// TwinCAT 3 PLC project PLC
// ProgramVersion: 3.1.4023.0
// libraries:
//   Tc2_Standard, * (Beckhoff Automation GmbH)
//   Tc2_System, * (Beckhoff Automation GmbH)
//   Tc3_Module, * (Beckhoff Automation GmbH)
// project tree:
//   / PlcTask.TcTTO
//   POUs/ MAIN.TcPOU
//   DUTs/IO/PdoEntries/ Status_3E6F3FF3.TcDUT, Control_6EF2C5D0.TcDUT, Status_237FCB0F.TcDUT, Setting_24C04940.TcDUT, Ctrl_56BB2DF2.TcDUT, Status_51F0A924.TcDUT, Settings_24C04940.TcDUT, Control_18D542D9.TcDUT, Status_396FCBA0.TcDUT, U1_STATUS_B0753356.TcDUT, U1_SAMPLES_2D13B74B.TcDUT, I1_STATUS_B0753356.TcDUT, I1_SAMPLES_2D13B74B.TcDUT, U2_STATUS_B0753356.TcDUT, U2_SAMPLES_2D13B74B.TcDUT, I2_STATUS_B0753356.TcDUT, I2_SAMPLES_2D13B74B.TcDUT, U3_STATUS_B0753356.TcDUT, U3_SAMPLES_2D13B74B.TcDUT, I3_STATUS_B0753356.TcDUT, I3_SAMPLES_2D13B74B.TcDUT, FSOE_31BB7F2A.TcDUT, FSOE_3C294B21.TcDUT, FSOE_13BCEA3F.TcDUT, FSOE_6A82EB93.TcDUT, FSOE_BB3344D6.TcDUT
//   DUTs/IO/PDOs/ InfoData_6F19DB2B.TcDUT, Channel_830843C1.TcDUT, Channel_42CA91F7.TcDUT, WcState_9091E0EB.TcDUT, DO_Diag_Inputs_CC455148.TcDUT, DO_Diag_Inputs_212B82C1.TcDUT, DO_Inputs_Device_AF161A9E.TcDUT, DO_Outputs_28AC1A9E.TcDUT, DO_Outputs_Device_36A5EF17.TcDUT, InfoData_32EB74EA.TcDUT, InfoData_0A66F009.TcDUT, ENC_Inputs_B3536485.TcDUT, ENC_Inputs_24B63C53.TcDUT, ENC_Outputs_21E2D14D.TcDUT, Ch1_CycleCount_9DBE2BC5.TcDUT, Ch1_Input_FFC4CE24.TcDUT, EMPTY_STRUCTURE.TcDUT, Ch2_CycleCount_976A51B5.TcDUT, Ch2_Input_78ADA90C.TcDUT, NextSync1Time_EE185E17.TcDUT, InfoData_A7436BC6.TcDUT, CycCount0_2C233804.TcDUT, Sample_0023574C.TcDUT, CycCount1_2C233804.TcDUT, Sample_07D5B44A.TcDUT, WcState_0B2B16F9.TcDUT, CycCount0_AF431CE0.TcDUT, CycCount1_A8B5FFE6.TcDUT, StartTimeNextOutput_228767F4.TcDUT, SAI_Inputs_3A838E11.TcDUT, SAI_Range_C3200E78.TcDUT, SAI_Range_3710D747.TcDUT, SAI_Inputs_84B29FE9.TcDUT, SAI_Range_BDBF6DA9.TcDUT, SAI_Range_2A187FC5.TcDUT, Channel_B90637B9.TcDUT, Channel_C6781B15.TcDUT, ENC_Inputs_3399C5AA.TcDUT, ENC_Outputs_2E45048F.TcDUT, ENC_Inputs_561E041F.TcDUT, ENC_Inputs_F139456B.TcDUT, ENC_Outputs_6FDDC669.TcDUT, L1_Voltage_Status_784F03AD.TcDUT, L1_Voltage_Samples_ED678DEE.TcDUT, L1_Current_Samples_89E07818.TcDUT, L1_Current_Samples_3209B12F.TcDUT, L2_Voltage_Status_0626A010.TcDUT, L2_Voltage_Samples_D91109BE.TcDUT, L2_Current_Status_F789DBA5.TcDUT, L2_Current_Samples_067F357F.TcDUT, L3_Voltage_Status_2C01C17B.TcDUT, L3_Voltage_Samples_CAC3758E.TcDUT, L3_Current_Status_DDAEBACE.TcDUT, L3_Current_Samples_15AD494F.TcDUT, AI_Timestamp_NextSync1Time_9AFDC275.TcDUT, AI_CycleCount_B1A935A2.TcDUT, InfoData_BEF6B88E.TcDUT, Digital_BD004D6F.TcDUT, Encoder_Channel_2E4EA213.TcDUT, Digital_A7E1DFAB.TcDUT, Analog_Channel_5F9B7EA6.TcDUT, Encoder_Channel_B7999E14.TcDUT, DeviceMain_Outputs_650F3486.TcDUT, FSoE_Slave_Connection_1_Slave_Message_330A35E4.TcDUT, Standard_Inputdata_FDD1436A.TcDUT, FSLOGIC_Inputs_CD3F9A93.TcDUT, FSoE_Slave_Connection_1_Master_Message_7109E4F0.TcDUT, Standard_Outputdata_59C030BE.TcDUT, Ch_A_AxisMain_Inputs_DC14661D.TcDUT, Ch_A_AxisMain_Outputs_A99AE12E.TcDUT, Ch_A_Interpolator_Outputs_462A5F1D.TcDUT, Ch_A_PositionControl_Inputs_8CB0F55A.TcDUT, WcState_B516A264.TcDUT, InfoData_358A59CF.TcDUT, Device_6E257577.TcDUT, Device_Safety_C21945A1.TcDUT, Ch_A_1FF86D85.TcDUT, Ch_A_AxisMain_Inputs_BA7CE8DB.TcDUT, Ch_A_D18C6F16.TcDUT, Ch_B_AxisMain_Inputs_A10B23CB.TcDUT, Ch_B_AxisMain_Outputs_526A47F8.TcDUT, Ch_B_Interpolator_Outputs_F819AE72.TcDUT, Ch_B_PositionControl_Inputs_C884000A.TcDUT, InfoData_386C00A5.TcDUT, Ch_B_5E084BAA.TcDUT, Ch_B_AxisMain_Inputs_3D4AF970.TcDUT, Ch_B_647F9A0C.TcDUT, InfoData_E68C61CD.TcDUT, InfoData_2A97D6CF.TcDUT, Inputs_25A0042B.TcDUT, Outputs_2397A10E.TcDUT
//   DUTs/IO/Boxes/ EK1100_1FC0878B.TcDUT, EK1122_1FC0878B.TcDUT, EPP2339_8DFD1558.TcDUT, EPP2349_8DFD1558.TcDUT, EP2316_3C060514.TcDUT, EP2338_39FFBC52.TcDUT, EP2339_C2A6198C.TcDUT, EP2339_56BCD6FB.TcDUT, EJ5151_905C5FD8.TcDUT, EL1262_0FA571DE.TcDUT, EL2262_79C970B1.TcDUT, EL2262_147DB6E1.TcDUT, EL2262_9619875D.TcDUT, EL3681_02A14E64.TcDUT, EL3681_0095B62C.TcDUT, EL5101_127DF9F1.TcDUT, EL5151_84FDBA5C.TcDUT, EL5151_93354628.TcDUT, EL5151_905C5FD8.TcDUT, EL5151_4D0E77FC.TcDUT, EL3773_D0D76902.TcDUT, EM7004_866015E1.TcDUT, AX8108_8297A621.TcDUT, AX8108_F7A82895.TcDUT, AX8118_8297A621.TcDUT, AX8118_F7A82895.TcDUT, AX8206_63F473B4.TcDUT, AX8206_FA9FF81E.TcDUT, AMP8000_F7A82895.TcDUT
//   DUTs/IO/Devices/ SyncUnitTask_2D604ED5.TcDUT, SyncUnitTasks_6FEB8257.TcDUT, SyncUnits_99E584AF.TcDUT
//   DUTs/IO/Topology/ boxesEK1122_B55A8AA2.TcDUT, boxes_17897972.TcDUT, EtherCAT_Master_Duplicates_CB89F35C.TcDUT
//   DUTs/IO/Base/ EtcSlaveBase_82538BE2.TcDUT, EtcSlaveBase_82538BE2.TcDUT, EtcSlaveBase_82538BE2.TcDUT, EtcSlaveTerminalBase_947E5A46.TcDUT, EtcSlaveBoxBase_77A0E4A7.TcDUT, EtcSlaveEndTerminalBase_866C7F0C.TcDUT, InputBase_8311D824.TcDUT, OutputBase_10CEE7DE.TcDUT, EtcMasterBase_62654B43.TcDUT
//   GVLs/ GVL_iXlinker.TcGVL

CONFIGURATION PLC
    RESOURCE PLC ON TwinCAT3
        TASK PlcTask(INTERVAL := T#10ms, PRIORITY := 20);
        PROGRAM MAIN WITH PlcTask : MAIN;
    END_RESOURCE
END_CONFIGURATION

// ---- DUTs/IO/PdoEntries/Status_3E6F3FF3.TcDUT
{attribute 'GeneratedUsingTerminal: EJ5151-0000-0016'}
{attribute addProperty BoxType "EJ5151-0000-0016"}
{attribute addProperty Id "Latch_C_validBOOL1Latch_extern_validBOOL1Set_counter_doneBOOL1Extrapolation_stallBOOL1Status_of_input_ABOOL1Status_of_input_BBOOL1Status_of_input_CBOOL1Status_of_extern_latchBOOL1Sync_errorBOOL1TxPDO_ToggleBOOL1"}
{attribute addProperty CRC "1047478259"}
{attribute addProperty Size "10"}
TYPE Status_3E6F3FF3 :
STRUCT
	{attribute addProperty Name "Latch_C_valid"}
	Latch_C_valid : BOOL;
	{attribute addProperty Name "Latch_extern_valid"}
	Latch_extern_valid : BOOL;
	{attribute addProperty Name "Set_counter_done"}
	Set_counter_done : BOOL;
	{attribute addProperty Name "Extrapolation_stall"}
	Extrapolation_stall : BOOL;
	{attribute addProperty Name "Status_of_input_A"}
	Status_of_input_A : BOOL;
	{attribute addProperty Name "Status_of_input_B"}
	Status_of_input_B : BOOL;
	{attribute addProperty Name "Status_of_input_C"}
	Status_of_input_C : BOOL;
	{attribute addProperty Name "Status_of_extern_latch"}
	Status_of_extern_latch : BOOL;
	{attribute addProperty Name "Sync_error"}
	Sync_error : BOOL;
	{attribute addProperty Name "TxPDO_Toggle"}
	TxPDO_Toggle : BOOL;
END_STRUCT
END_TYPE

// ---- DUTs/IO/PdoEntries/Control_6EF2C5D0.TcDUT
{attribute 'GeneratedUsingTerminal: EJ5151-0000-0016'}
{attribute addProperty BoxType "EJ5151-0000-0016"}
{attribute addProperty Id "Enable_latch_CBOOL1Enable_latch_extern_on_positive_edgeBOOL1Set_counterBOOL1Enable_latch_extern_on_negative_edgeBOOL1"}
{attribute addProperty CRC "1861404112"}
{attribute addProperty Size "4"}
TYPE Control_6EF2C5D0 :
STRUCT
	{attribute addProperty Name "Enable_latch_C"}
	Enable_latch_C : BOOL;
	{attribute addProperty Name "Enable_latch_extern_on_positive_edge"}
	Enable_latch_extern_on_positive_edge : BOOL;
	{attribute addProperty Name "Set_counter"}
	Set_counter : BOOL;
	{attribute addProperty Name "Enable_latch_extern_on_negative_edge"}
	Enable_latch_extern_on_negative_edge : BOOL;
END_STRUCT
END_TYPE

// ---- DUTs/IO/PdoEntries/Status_237FCB0F.TcDUT
{attribute 'GeneratedUsingTerminal: EL3681-0000-0017'}
{attribute addProperty BoxType "EL3681-0000-0017"}
{attribute addProperty Id "UnderrangeBOOL1OverrangeBOOL1Extended_rangeBOOL1Data_InvalidBOOL1Range_InvalidBOOL1Autorange_enabledBOOL1ErrorBOOL1Calibration_in_progressBOOL1TxPDO_StateBOOL1TxPDO_ToggleBOOL1"}
{attribute addProperty CRC "595577615"}
{attribute addProperty Size "10"}
TYPE Status_237FCB0F :
STRUCT
	{attribute addProperty Name "Underrange"}
	Underrange : BOOL;
	{attribute addProperty Name "Overrange"}
	Overrange : BOOL;
	{attribute addProperty Name "Extended_range"}
	Extended_range : BOOL;
	{attribute addProperty Name "Data_Invalid"}
	Data_Invalid : BOOL;
	{attribute addProperty Name "Range_Invalid"}
	Range_Invalid : BOOL;
	{attribute addProperty Name "Autorange_enabled"}
	Autorange_enabled : BOOL;
	{attribute addProperty Name "Error"}
	Error : BOOL;
	{attribute addProperty Name "Calibration_in_progress"}
	Calibration_in_progress : BOOL;
	{attribute addProperty Name "TxPDO_State"}
	TxPDO_State : BOOL;
	{attribute addProperty Name "TxPDO_Toggle"}
	TxPDO_Toggle : BOOL;
END_STRUCT
END_TYPE

// ---- DUTs/IO/PdoEntries/Setting_24C04940.TcDUT
{attribute 'GeneratedUsingTerminal: EL3681-0000-0017'}
{attribute addProperty BoxType "EL3681-0000-0017"}
{attribute addProperty Id "ModeBYTE1RangeSINT1"}
{attribute addProperty CRC "616581440"}
{attribute addProperty Size "2"}
TYPE Setting_24C04940 :
STRUCT
	{attribute addProperty Name "Mode"}
	Mode : BYTE;
	{attribute addProperty Name "Range"}
	Range : SINT;
END_STRUCT
END_TYPE

// ---- DUTs/IO/PdoEntries/Ctrl_56BB2DF2.TcDUT
{attribute 'GeneratedUsingTerminal: EL3681-0000-0017'}
{attribute addProperty BoxType "EL3681-0000-0017"}
{attribute addProperty Id "Enable_autorangeBOOL1ModeBYTE1RangeSINT1"}
{attribute addProperty CRC "1455107570"}
{attribute addProperty Size "3"}
TYPE Ctrl_56BB2DF2 :
STRUCT
	{attribute addProperty Name "Enable_autorange"}
	Enable_autorange : BOOL;
	{attribute addProperty Name "Mode"}
	Mode : BYTE;
	{attribute addProperty Name "Range"}
	Range : SINT;
END_STRUCT
END_TYPE

// ---- DUTs/IO/PdoEntries/Status_51F0A924.TcDUT
{attribute 'GeneratedUsingTerminal: EL3681-0000-0018'}
{attribute addProperty BoxType "EL3681-0000-0018"}
{attribute addProperty Id "UnderrangeBOOL1OverrangeBOOL1Extended_rangeBOOL1Data_invalidBOOL1Range_invalidBOOL1Autorange_disabledBOOL1ErrorBOOL1Calibration_in_progressBOOL1TxPDO_StateBOOL1TxPDO_ToggleBOOL1"}
{attribute addProperty CRC "1374726436"}
{attribute addProperty Size "10"}
TYPE Status_51F0A924 :
STRUCT
	{attribute addProperty Name "Underrange"}
	Underrange : BOOL;
	{attribute addProperty Name "Overrange"}
	Overrange : BOOL;
	{attribute addProperty Name "Extended_range"}
	Extended_range : BOOL;
	{attribute addProperty Name "Data_invalid"}
	Data_invalid : BOOL;
	{attribute addProperty Name "Range_invalid"}
	Range_invalid : BOOL;
	{attribute addProperty Name "Autorange_disabled"}
	Autorange_disabled : BOOL;
	{attribute addProperty Name "Error"}
	Error : BOOL;
	{attribute addProperty Name "Calibration_in_progress"}
	Calibration_in_progress : BOOL;
	{attribute addProperty Name "TxPDO_State"}
	TxPDO_State : BOOL;
	{attribute addProperty Name "TxPDO_Toggle"}
	TxPDO_Toggle : BOOL;
END_STRUCT
END_TYPE

// ---- DUTs/IO/PdoEntries/Settings_24C04940.TcDUT
{attribute 'GeneratedUsingTerminal: EL3681-0000-0018'}
{attribute addProperty BoxType "EL3681-0000-0018"}
{attribute addProperty Id "ModeBYTE1RangeSINT1"}
{attribute addProperty CRC "616581440"}
{attribute addProperty Size "2"}
TYPE Settings_24C04940 :
STRUCT
	{attribute addProperty Name "Mode"}
	Mode : BYTE;
	{attribute addProperty Name "Range"}
	Range : SINT;
END_STRUCT
END_TYPE

// ---- DUTs/IO/PdoEntries/Control_18D542D9.TcDUT
{attribute 'GeneratedUsingTerminal: EL3681-0000-0018'}
{attribute addProperty BoxType "EL3681-0000-0018"}
{attribute addProperty Id "Disable_autorangeBOOL1Start_calibrationBOOL1ModeBYTE1RangeSINT1"}
{attribute addProperty CRC "416629465"}
{attribute addProperty Size "4"}
TYPE Control_18D542D9 :
STRUCT
	{attribute addProperty Name "Disable_autorange"}
	Disable_autorange : BOOL;
	{attribute addProperty Name "Start_calibration"}
	Start_calibration : BOOL;
	{attribute addProperty Name "Mode"}
	Mode : BYTE;
	{attribute addProperty Name "Range"}
	Range : SINT;
END_STRUCT
END_TYPE

// ---- DUTs/IO/PdoEntries/Status_396FCBA0.TcDUT
{attribute 'GeneratedUsingTerminal: EL5151-0000-0016'}
{attribute addProperty BoxType "EL5151-0000-0016"}
{attribute addProperty Id "Latch_C_validBOOL1Latch_extern_validBOOL1Set_counter_doneBOOL1Status_of_input_ABOOL1Status_of_input_BBOOL1Status_of_input_CBOOL1Status_of_extern_latchBOOL1TxPDO_ToggleBOOL1"}
{attribute addProperty CRC "963627936"}
{attribute addProperty Size "8"}
TYPE Status_396FCBA0 :
STRUCT
	{attribute addProperty Name "Latch_C_valid"}
	Latch_C_valid : BOOL;
	{attribute addProperty Name "Latch_extern_valid"}
	Latch_extern_valid : BOOL;
	{attribute addProperty Name "Set_counter_done"}
	Set_counter_done : BOOL;
	{attribute addProperty Name "Status_of_input_A"}
	Status_of_input_A : BOOL;
	{attribute addProperty Name "Status_of_input_B"}
	Status_of_input_B : BOOL;
	{attribute addProperty Name "Status_of_input_C"}
	Status_of_input_C : BOOL;
	{attribute addProperty Name "Status_of_extern_latch"}
	Status_of_extern_latch : BOOL;
	{attribute addProperty Name "TxPDO_Toggle"}
	TxPDO_Toggle : BOOL;
END_STRUCT
END_TYPE

// ---- DUTs/IO/PdoEntries/U1_STATUS_B0753356.TcDUT
{attribute 'GeneratedUsingTerminal: EL3773-0000-0016'}
{attribute addProperty BoxType "EL3773-0000-0016"}
{attribute addProperty Id "UnderrangeBOOL1OverrangeBOOL1Limit_1BYTE1Limit_2BYTE1ErrorBOOL1Sync_errorBOOL1TxPDO_StateBOOL1TxPDO_ToggleBOOL1"}
{attribute addProperty CRC "2960470870"}
{attribute addProperty Size "8"}
TYPE U1_STATUS_B0753356 :
STRUCT
	{attribute addProperty Name "Underrange"}
	Underrange : BOOL;
	{attribute addProperty Name "Overrange"}
	Overrange : BOOL;
	{attribute addProperty Name "Limit_1"}
	Limit_1 : BYTE;
	{attribute addProperty Name "Limit_2"}
	Limit_2 : BYTE;
	{attribute addProperty Name "Error"}
	Error : BOOL;
	{attribute addProperty Name "Sync_error"}
	Sync_error : BOOL;
	{attribute addProperty Name "TxPDO_State"}
	TxPDO_State : BOOL;
	{attribute addProperty Name "TxPDO_Toggle"}
	TxPDO_Toggle : BOOL;
END_STRUCT
END_TYPE

// ---- DUTs/IO/PdoEntries/U1_SAMPLES_2D13B74B.TcDUT
{attribute 'GeneratedUsingTerminal: EL3773-0000-0016'}
{attribute addProperty BoxType "EL3773-0000-0016"}
{attribute addProperty Id "Sample_1INT2Sample_2INT2Sample_3INT2Sample_4INT2Sample_5INT2Sample_6INT2Sample_7INT2Sample_8INT2Sample_9INT2Sample_10INT2"}
{attribute addProperty CRC "756266827"}
{attribute addProperty Size "20"}
TYPE U1_SAMPLES_2D13B74B :
STRUCT
	{attribute addProperty Name "Sample_1"}
	Sample_1 : INT;
	{attribute addProperty Name "Sample_2"}
	Sample_2 : INT;
	{attribute addProperty Name "Sample_3"}
	Sample_3 : INT;
	{attribute addProperty Name "Sample_4"}
	Sample_4 : INT;
	{attribute addProperty Name "Sample_5"}
	Sample_5 : INT;
	{attribute addProperty Name "Sample_6"}
	Sample_6 : INT;
	{attribute addProperty Name "Sample_7"}
	Sample_7 : INT;
	{attribute addProperty Name "Sample_8"}
	Sample_8 : INT;
	{attribute addProperty Name "Sample_9"}
	Sample_9 : INT;
	{attribute addProperty Name "Sample_10"}
	Sample_10 : INT;
END_STRUCT
END_TYPE

// ---- DUTs/IO/PdoEntries/I1_STATUS_B0753356.TcDUT
{attribute 'GeneratedUsingTerminal: EL3773-0000-0016'}
{attribute addProperty BoxType "EL3773-0000-0016"}
{attribute addProperty Id "UnderrangeBOOL1OverrangeBOOL1Limit_1BYTE1Limit_2BYTE1ErrorBOOL1Sync_errorBOOL1TxPDO_StateBOOL1TxPDO_ToggleBOOL1"}
{attribute addProperty CRC "2960470870"}
{attribute addProperty Size "8"}
TYPE I1_STATUS_B0753356 :
STRUCT
	{attribute addProperty Name "Underrange"}
	Underrange : BOOL;
	{attribute addProperty Name "Overrange"}
	Overrange : BOOL;
	{attribute addProperty Name "Limit_1"}
	Limit_1 : BYTE;
	{attribute addProperty Name "Limit_2"}
	Limit_2 : BYTE;
	{attribute addProperty Name "Error"}
	Error : BOOL;
	{attribute addProperty Name "Sync_error"}
	Sync_error : BOOL;
	{attribute addProperty Name "TxPDO_State"}
	TxPDO_State : BOOL;
	{attribute addProperty Name "TxPDO_Toggle"}
	TxPDO_Toggle : BOOL;
END_STRUCT
END_TYPE

// ---- DUTs/IO/PdoEntries/I1_SAMPLES_2D13B74B.TcDUT
{attribute 'GeneratedUsingTerminal: EL3773-0000-0016'}
{attribute addProperty BoxType "EL3773-0000-0016"}
{attribute addProperty Id "Sample_1INT2Sample_2INT2Sample_3INT2Sample_4INT2Sample_5INT2Sample_6INT2Sample_7INT2Sample_8INT2Sample_9INT2Sample_10INT2"}
{attribute addProperty CRC "756266827"}
{attribute addProperty Size "20"}
TYPE I1_SAMPLES_2D13B74B :
STRUCT
	{attribute addProperty Name "Sample_1"}
	Sample_1 : INT;
	{attribute addProperty Name "Sample_2"}
	Sample_2 : INT;
	{attribute addProperty Name "Sample_3"}
	Sample_3 : INT;
	{attribute addProperty Name "Sample_4"}
	Sample_4 : INT;
	{attribute addProperty Name "Sample_5"}
	Sample_5 : INT;
	{attribute addProperty Name "Sample_6"}
	Sample_6 : INT;
	{attribute addProperty Name "Sample_7"}
	Sample_7 : INT;
	{attribute addProperty Name "Sample_8"}
	Sample_8 : INT;
	{attribute addProperty Name "Sample_9"}
	Sample_9 : INT;
	{attribute addProperty Name "Sample_10"}
	Sample_10 : INT;
END_STRUCT
END_TYPE

// ---- DUTs/IO/PdoEntries/U2_STATUS_B0753356.TcDUT
{attribute 'GeneratedUsingTerminal: EL3773-0000-0016'}
{attribute addProperty BoxType "EL3773-0000-0016"}
{attribute addProperty Id "UnderrangeBOOL1OverrangeBOOL1Limit_1BYTE1Limit_2BYTE1ErrorBOOL1Sync_errorBOOL1TxPDO_StateBOOL1TxPDO_ToggleBOOL1"}
{attribute addProperty CRC "2960470870"}
{attribute addProperty Size "8"}
TYPE U2_STATUS_B0753356 :
STRUCT
	{attribute addProperty Name "Underrange"}
	Underrange : BOOL;
	{attribute addProperty Name "Overrange"}
	Overrange : BOOL;
	{attribute addProperty Name "Limit_1"}
	Limit_1 : BYTE;
	{attribute addProperty Name "Limit_2"}
	Limit_2 : BYTE;
	{attribute addProperty Name "Error"}
	Error : BOOL;
	{attribute addProperty Name "Sync_error"}
	Sync_error : BOOL;
	{attribute addProperty Name "TxPDO_State"}
	TxPDO_State : BOOL;
	{attribute addProperty Name "TxPDO_Toggle"}
	TxPDO_Toggle : BOOL;
END_STRUCT
END_TYPE

// ---- DUTs/IO/PdoEntries/U2_SAMPLES_2D13B74B.TcDUT
{attribute 'GeneratedUsingTerminal: EL3773-0000-0016'}
{attribute addProperty BoxType "EL3773-0000-0016"}
{attribute addProperty Id "Sample_1INT2Sample_2INT2Sample_3INT2Sample_4INT2Sample_5INT2Sample_6INT2Sample_7INT2Sample_8INT2Sample_9INT2Sample_10INT2"}
{attribute addProperty CRC "756266827"}
{attribute addProperty Size "20"}
TYPE U2_SAMPLES_2D13B74B :
STRUCT
	{attribute addProperty Name "Sample_1"}
	Sample_1 : INT;
	{attribute addProperty Name "Sample_2"}
	Sample_2 : INT;
	{attribute addProperty Name "Sample_3"}
	Sample_3 : INT;
	{attribute addProperty Name "Sample_4"}
	Sample_4 : INT;
	{attribute addProperty Name "Sample_5"}
	Sample_5 : INT;
	{attribute addProperty Name "Sample_6"}
	Sample_6 : INT;
	{attribute addProperty Name "Sample_7"}
	Sample_7 : INT;
	{attribute addProperty Name "Sample_8"}
	Sample_8 : INT;
	{attribute addProperty Name "Sample_9"}
	Sample_9 : INT;
	{attribute addProperty Name "Sample_10"}
	Sample_10 : INT;
END_STRUCT
END_TYPE

// ---- DUTs/IO/PdoEntries/I2_STATUS_B0753356.TcDUT
{attribute 'GeneratedUsingTerminal: EL3773-0000-0016'}
{attribute addProperty BoxType "EL3773-0000-0016"}
{attribute addProperty Id "UnderrangeBOOL1OverrangeBOOL1Limit_1BYTE1Limit_2BYTE1ErrorBOOL1Sync_errorBOOL1TxPDO_StateBOOL1TxPDO_ToggleBOOL1"}
{attribute addProperty CRC "2960470870"}
{attribute addProperty Size "8"}
TYPE I2_STATUS_B0753356 :
STRUCT
	{attribute addProperty Name "Underrange"}
	Underrange : BOOL;
	{attribute addProperty Name "Overrange"}
	Overrange : BOOL;
	{attribute addProperty Name "Limit_1"}
	Limit_1 : BYTE;
	{attribute addProperty Name "Limit_2"}
	Limit_2 : BYTE;
	{attribute addProperty Name "Error"}
	Error : BOOL;
	{attribute addProperty Name "Sync_error"}
	Sync_error : BOOL;
	{attribute addProperty Name "TxPDO_State"}
	TxPDO_State : BOOL;
	{attribute addProperty Name "TxPDO_Toggle"}
	TxPDO_Toggle : BOOL;
END_STRUCT
END_TYPE

// ---- DUTs/IO/PdoEntries/I2_SAMPLES_2D13B74B.TcDUT
{attribute 'GeneratedUsingTerminal: EL3773-0000-0016'}
{attribute addProperty BoxType "EL3773-0000-0016"}
{attribute addProperty Id "Sample_1INT2Sample_2INT2Sample_3INT2Sample_4INT2Sample_5INT2Sample_6INT2Sample_7INT2Sample_8INT2Sample_9INT2Sample_10INT2"}
{attribute addProperty CRC "756266827"}
{attribute addProperty Size "20"}
TYPE I2_SAMPLES_2D13B74B :
STRUCT
	{attribute addProperty Name "Sample_1"}
	Sample_1 : INT;
	{attribute addProperty Name "Sample_2"}
	Sample_2 : INT;
	{attribute addProperty Name "Sample_3"}
	Sample_3 : INT;
	{attribute addProperty Name "Sample_4"}
	Sample_4 : INT;
	{attribute addProperty Name "Sample_5"}
	Sample_5 : INT;
	{attribute addProperty Name "Sample_6"}
	Sample_6 : INT;
	{attribute addProperty Name "Sample_7"}
	Sample_7 : INT;
	{attribute addProperty Name "Sample_8"}
	Sample_8 : INT;
	{attribute addProperty Name "Sample_9"}
	Sample_9 : INT;
	{attribute addProperty Name "Sample_10"}
	Sample_10 : INT;
END_STRUCT
END_TYPE

// ---- DUTs/IO/PdoEntries/U3_STATUS_B0753356.TcDUT
{attribute 'GeneratedUsingTerminal: EL3773-0000-0016'}
{attribute addProperty BoxType "EL3773-0000-0016"}
{attribute addProperty Id "UnderrangeBOOL1OverrangeBOOL1Limit_1BYTE1Limit_2BYTE1ErrorBOOL1Sync_errorBOOL1TxPDO_StateBOOL1TxPDO_ToggleBOOL1"}
{attribute addProperty CRC "2960470870"}
{attribute addProperty Size "8"}
TYPE U3_STATUS_B0753356 :
STRUCT
	{attribute addProperty Name "Underrange"}
	Underrange : BOOL;
	{attribute addProperty Name "Overrange"}
	Overrange : BOOL;
	{attribute addProperty Name "Limit_1"}
	Limit_1 : BYTE;
	{attribute addProperty Name "Limit_2"}
	Limit_2 : BYTE;
	{attribute addProperty Name "Error"}
	Error : BOOL;
	{attribute addProperty Name "Sync_error"}
	Sync_error : BOOL;
	{attribute addProperty Name "TxPDO_State"}
	TxPDO_State : BOOL;
	{attribute addProperty Name "TxPDO_Toggle"}
	TxPDO_Toggle : BOOL;
END_STRUCT
END_TYPE

// ---- DUTs/IO/PdoEntries/U3_SAMPLES_2D13B74B.TcDUT
{attribute 'GeneratedUsingTerminal: EL3773-0000-0016'}
{attribute addProperty BoxType "EL3773-0000-0016"}
{attribute addProperty Id "Sample_1INT2Sample_2INT2Sample_3INT2Sample_4INT2Sample_5INT2Sample_6INT2Sample_7INT2Sample_8INT2Sample_9INT2Sample_10INT2"}
{attribute addProperty CRC "756266827"}
{attribute addProperty Size "20"}
TYPE U3_SAMPLES_2D13B74B :
STRUCT
	{attribute addProperty Name "Sample_1"}
	Sample_1 : INT;
	{attribute addProperty Name "Sample_2"}
	Sample_2 : INT;
	{attribute addProperty Name "Sample_3"}
	Sample_3 : INT;
	{attribute addProperty Name "Sample_4"}
	Sample_4 : INT;
	{attribute addProperty Name "Sample_5"}
	Sample_5 : INT;
	{attribute addProperty Name "Sample_6"}
	Sample_6 : INT;
	{attribute addProperty Name "Sample_7"}
	Sample_7 : INT;
	{attribute addProperty Name "Sample_8"}
	Sample_8 : INT;
	{attribute addProperty Name "Sample_9"}
	Sample_9 : INT;
	{attribute addProperty Name "Sample_10"}
	Sample_10 : INT;
END_STRUCT
END_TYPE

// ---- DUTs/IO/PdoEntries/I3_STATUS_B0753356.TcDUT
{attribute 'GeneratedUsingTerminal: EL3773-0000-0016'}
{attribute addProperty BoxType "EL3773-0000-0016"}
{attribute addProperty Id "UnderrangeBOOL1OverrangeBOOL1Limit_1BYTE1Limit_2BYTE1ErrorBOOL1Sync_errorBOOL1TxPDO_StateBOOL1TxPDO_ToggleBOOL1"}
{attribute addProperty CRC "2960470870"}
{attribute addProperty Size "8"}
TYPE I3_STATUS_B0753356 :
STRUCT
	{attribute addProperty Name "Underrange"}
	Underrange : BOOL;
	{attribute addProperty Name "Overrange"}
	Overrange : BOOL;
	{attribute addProperty Name "Limit_1"}
	Limit_1 : BYTE;
	{attribute addProperty Name "Limit_2"}
	Limit_2 : BYTE;
	{attribute addProperty Name "Error"}
	Error : BOOL;
	{attribute addProperty Name "Sync_error"}
	Sync_error : BOOL;
	{attribute addProperty Name "TxPDO_State"}
	TxPDO_State : BOOL;
	{attribute addProperty Name "TxPDO_Toggle"}
	TxPDO_Toggle : BOOL;
END_STRUCT
END_TYPE

// ---- DUTs/IO/PdoEntries/I3_SAMPLES_2D13B74B.TcDUT
{attribute 'GeneratedUsingTerminal: EL3773-0000-0016'}
{attribute addProperty BoxType "EL3773-0000-0016"}
{attribute addProperty Id "Sample_1INT2Sample_2INT2Sample_3INT2Sample_4INT2Sample_5INT2Sample_6INT2Sample_7INT2Sample_8INT2Sample_9INT2Sample_10INT2"}
{attribute addProperty CRC "756266827"}
{attribute addProperty Size "20"}
TYPE I3_SAMPLES_2D13B74B :
STRUCT
	{attribute addProperty Name "Sample_1"}
	Sample_1 : INT;
	{attribute addProperty Name "Sample_2"}
	Sample_2 : INT;
	{attribute addProperty Name "Sample_3"}
	Sample_3 : INT;
	{attribute addProperty Name "Sample_4"}
	Sample_4 : INT;
	{attribute addProperty Name "Sample_5"}
	Sample_5 : INT;
	{attribute addProperty Name "Sample_6"}
	Sample_6 : INT;
	{attribute addProperty Name "Sample_7"}
	Sample_7 : INT;
	{attribute addProperty Name "Sample_8"}
	Sample_8 : INT;
	{attribute addProperty Name "Sample_9"}
	Sample_9 : INT;
	{attribute addProperty Name "Sample_10"}
	Sample_10 : INT;
END_STRUCT
END_TYPE

// ---- DUTs/IO/PdoEntries/FSOE_31BB7F2A.TcDUT
{attribute 'GeneratedUsingTerminal: AX8108-0100-0101-0101'}
{attribute addProperty BoxType "AX8108-0100-0101-0101"}
{attribute addProperty Id "FSoE_Slave_CmdUSINT1Axis_A_STOBOOL1Safe_Input_1BOOL1Safe_Input_2BOOL1Safe_Input_3BOOL1Safe_Input_4BOOL1Safe_Input_5BOOL1Safe_Input_6BOOL1Safe_Input_7BOOL1Axis_B_STOBOOL1Safe_Input_9BOOL1Safe_Input_10BOOL1Safe_Input_11BOOL1Safe_Input_12BOOL1Safe_Input_13BOOL1Safe_Input_14BOOL1Safe_Input_15BOOL1FSoE_Slave_CRC_0UINT2FSoE_Slave_ConnIDUINT2"}
{attribute addProperty CRC "834371370"}
{attribute addProperty Size "21"}
TYPE FSOE_31BB7F2A :
STRUCT
	{attribute addProperty Name "FSoE_Slave_Cmd"}
	FSoE_Slave_Cmd : USINT;
	{attribute addProperty Name "Axis_A_STO"}
	Axis_A_STO : BOOL;
	{attribute addProperty Name "Safe_Input_1"}
	Safe_Input_1 : BOOL;
	{attribute addProperty Name "Safe_Input_2"}
	Safe_Input_2 : BOOL;
	{attribute addProperty Name "Safe_Input_3"}
	Safe_Input_3 : BOOL;
	{attribute addProperty Name "Safe_Input_4"}
	Safe_Input_4 : BOOL;
	{attribute addProperty Name "Safe_Input_5"}
	Safe_Input_5 : BOOL;
	{attribute addProperty Name "Safe_Input_6"}
	Safe_Input_6 : BOOL;
	{attribute addProperty Name "Safe_Input_7"}
	Safe_Input_7 : BOOL;
	{attribute addProperty Name "Axis_B_STO"}
	Axis_B_STO : BOOL;
	{attribute addProperty Name "Safe_Input_9"}
	Safe_Input_9 : BOOL;
	{attribute addProperty Name "Safe_Input_10"}
	Safe_Input_10 : BOOL;
	{attribute addProperty Name "Safe_Input_11"}
	Safe_Input_11 : BOOL;
	{attribute addProperty Name "Safe_Input_12"}
	Safe_Input_12 : BOOL;
	{attribute addProperty Name "Safe_Input_13"}
	Safe_Input_13 : BOOL;
	{attribute addProperty Name "Safe_Input_14"}
	Safe_Input_14 : BOOL;
	{attribute addProperty Name "Safe_Input_15"}
	Safe_Input_15 : BOOL;
	{attribute addProperty Name "FSoE_Slave_CRC_0"}
	FSoE_Slave_CRC_0 : UINT;
	{attribute addProperty Name "FSoE_Slave_ConnID"}
	FSoE_Slave_ConnID : UINT;
END_STRUCT
END_TYPE

// ---- DUTs/IO/PdoEntries/FSOE_3C294B21.TcDUT
{attribute 'GeneratedUsingTerminal: AX8108-0100-0101-0101'}
{attribute addProperty BoxType "AX8108-0100-0101-0101"}
{attribute addProperty Id "Std_InputBOOL1Std_Input_1BOOL1Std_Input_2BOOL1Std_Input_3BOOL1Std_Input_4BOOL1Std_Input_5BOOL1Std_Input_6BOOL1Std_Input_7BOOL1"}
{attribute addProperty CRC "1009339169"}
{attribute addProperty Size "8"}
TYPE FSOE_3C294B21 :
STRUCT
	{attribute addProperty Name "Std_Input"}
	Std_Input : BOOL;
	{attribute addProperty Name "Std_Input_1"}
	Std_Input_1 : BOOL;
	{attribute addProperty Name "Std_Input_2"}
	Std_Input_2 : BOOL;
	{attribute addProperty Name "Std_Input_3"}
	Std_Input_3 : BOOL;
	{attribute addProperty Name "Std_Input_4"}
	Std_Input_4 : BOOL;
	{attribute addProperty Name "Std_Input_5"}
	Std_Input_5 : BOOL;
	{attribute addProperty Name "Std_Input_6"}
	Std_Input_6 : BOOL;
	{attribute addProperty Name "Std_Input_7"}
	Std_Input_7 : BOOL;
END_STRUCT
END_TYPE

// ---- DUTs/IO/PdoEntries/FSOE_13BCEA3F.TcDUT
{attribute 'GeneratedUsingTerminal: AX8108-0100-0101-0101'}
{attribute addProperty BoxType "AX8108-0100-0101-0101"}
{attribute addProperty Id "Safe_Logic_StateUSINT1Cycle_CounterUSINT1"}
{attribute addProperty CRC "331147839"}
{attribute addProperty Size "2"}
TYPE FSOE_13BCEA3F :
STRUCT
	{attribute addProperty Name "Safe_Logic_State"}
	Safe_Logic_State : USINT;
	{attribute addProperty Name "Cycle_Counter"}
	Cycle_Counter : USINT;
END_STRUCT
END_TYPE

// ---- DUTs/IO/PdoEntries/FSOE_6A82EB93.TcDUT
{attribute 'GeneratedUsingTerminal: AX8108-0100-0101-0101'}
{attribute addProperty BoxType "AX8108-0100-0101-0101"}
{attribute addProperty Id "FSoE_Master_CmdUSINT1Axis_A_STOBOOL1Safe_Output_1BOOL1Safe_Output_2BOOL1Safe_Output_3BOOL1Safe_Output_4BOOL1Safe_Output_5BOOL1Safe_Output_6BOOL1Safe_Output_7BOOL1Axis_B_STOBOOL1Safe_Output_9BOOL1Safe_Output_10BOOL1Safe_Output_11BOOL1Safe_Output_12BOOL1Safe_Output_13BOOL1Safe_Output_14BOOL1Safe_Output_15BOOL1FSoE_Master_CRC_0UINT2FSoE_Master_ConnIDUINT2"}
{attribute addProperty CRC "1786964883"}
{attribute addProperty Size "21"}
TYPE FSOE_6A82EB93 :
STRUCT
	{attribute addProperty Name "FSoE_Master_Cmd"}
	FSoE_Master_Cmd : USINT;
	{attribute addProperty Name "Axis_A_STO"}
	Axis_A_STO : BOOL;
	{attribute addProperty Name "Safe_Output_1"}
	Safe_Output_1 : BOOL;
	{attribute addProperty Name "Safe_Output_2"}
	Safe_Output_2 : BOOL;
	{attribute addProperty Name "Safe_Output_3"}
	Safe_Output_3 : BOOL;
	{attribute addProperty Name "Safe_Output_4"}
	Safe_Output_4 : BOOL;
	{attribute addProperty Name "Safe_Output_5"}
	Safe_Output_5 : BOOL;
	{attribute addProperty Name "Safe_Output_6"}
	Safe_Output_6 : BOOL;
	{attribute addProperty Name "Safe_Output_7"}
	Safe_Output_7 : BOOL;
	{attribute addProperty Name "Axis_B_STO"}
	Axis_B_STO : BOOL;
	{attribute addProperty Name "Safe_Output_9"}
	Safe_Output_9 : BOOL;
	{attribute addProperty Name "Safe_Output_10"}
	Safe_Output_10 : BOOL;
	{attribute addProperty Name "Safe_Output_11"}
	Safe_Output_11 : BOOL;
	{attribute addProperty Name "Safe_Output_12"}
	Safe_Output_12 : BOOL;
	{attribute addProperty Name "Safe_Output_13"}
	Safe_Output_13 : BOOL;
	{attribute addProperty Name "Safe_Output_14"}
	Safe_Output_14 : BOOL;
	{attribute addProperty Name "Safe_Output_15"}
	Safe_Output_15 : BOOL;
	{attribute addProperty Name "FSoE_Master_CRC_0"}
	FSoE_Master_CRC_0 : UINT;
	{attribute addProperty Name "FSoE_Master_ConnID"}
	FSoE_Master_ConnID : UINT;
END_STRUCT
END_TYPE

// ---- DUTs/IO/PdoEntries/FSOE_BB3344D6.TcDUT
{attribute 'GeneratedUsingTerminal: AX8108-0100-0101-0101'}
{attribute addProperty BoxType "AX8108-0100-0101-0101"}
{attribute addProperty Id "Std_OutputBOOL1Std_Output_1BOOL1Std_Output_2BOOL1Std_Output_3BOOL1Std_Output_4BOOL1Std_Output_5BOOL1Std_Output_6BOOL1Std_Output_7BOOL1"}
{attribute addProperty CRC "3140699350"}
{attribute addProperty Size "8"}
TYPE FSOE_BB3344D6 :
STRUCT
	{attribute addProperty Name "Std_Output"}
	Std_Output : BOOL;
	{attribute addProperty Name "Std_Output_1"}
	Std_Output_1 : BOOL;
	{attribute addProperty Name "Std_Output_2"}
	Std_Output_2 : BOOL;
	{attribute addProperty Name "Std_Output_3"}
	Std_Output_3 : BOOL;
	{attribute addProperty Name "Std_Output_4"}
	Std_Output_4 : BOOL;
	{attribute addProperty Name "Std_Output_5"}
	Std_Output_5 : BOOL;
	{attribute addProperty Name "Std_Output_6"}
	Std_Output_6 : BOOL;
	{attribute addProperty Name "Std_Output_7"}
	Std_Output_7 : BOOL;
END_STRUCT
END_TYPE

// ---- DUTs/IO/PDOs/InfoData_6F19DB2B.TcDUT
{attribute 'GeneratedUsingTerminal: EK1100-0000-0018'}
{attribute addProperty BoxType "EK1100-0000-0018"}
{attribute addProperty Id "StateAT %I*UINT2"}
{attribute addProperty CRC "1863965483"}
{attribute addProperty Size "2"}
TYPE InfoData_6F19DB2B :
STRUCT
	{attribute addProperty Name "State"}
	State AT %I* : UINT;
END_STRUCT
END_TYPE

// ---- DUTs/IO/PDOs/Channel_830843C1.TcDUT
{attribute 'GeneratedUsingTerminal: EPP2339-0021-0016'}
{attribute addProperty BoxType "EPP2339-0021-0016"}
{attribute addProperty Id "InputAT %I*BOOL1"}
{attribute addProperty CRC "2198356929"}
{attribute addProperty Size "1"}
TYPE Channel_830843C1 EXTENDS InputBase_8311D824 :
STRUCT
	{attribute addProperty Name "Input"}
	Input AT %I* : BOOL;
END_STRUCT
END_TYPE

// ---- DUTs/IO/PDOs/Channel_42CA91F7.TcDUT
{attribute 'GeneratedUsingTerminal: EPP2339-0021-0016'}
{attribute addProperty BoxType "EPP2339-0021-0016"}
{attribute addProperty Id "OutputAT %Q*BOOL1"}
{attribute addProperty CRC "1120571895"}
{attribute addProperty Size "1"}
TYPE Channel_42CA91F7 EXTENDS OutputBase_10CEE7DE :
STRUCT
	{attribute addProperty Name "Output"}
	Output AT %Q* : BOOL;
END_STRUCT
END_TYPE

// ---- DUTs/IO/PDOs/WcState_9091E0EB.TcDUT
{attribute 'GeneratedUsingTerminal: EPP2339-0021-0016'}
{attribute addProperty BoxType "EPP2339-0021-0016"}
{attribute addProperty Id "WcStateAT %I*BOOL1InputToggleAT %I*BOOL1"}
{attribute addProperty CRC "2425479403"}
{attribute addProperty Size "2"}
TYPE WcState_9091E0EB :
STRUCT
	{attribute addProperty Name "WcState"}
	WcState AT %I* : BOOL;
	{attribute addProperty Name "InputToggle"}
	InputToggle AT %I* : BOOL;
END_STRUCT
END_TYPE

// ---- DUTs/IO/PDOs/DO_Diag_Inputs_CC455148.TcDUT
{attribute 'GeneratedUsingTerminal: EP2316-0008-0017'}
{attribute addProperty BoxType "EP2316-0008-0017"}
{attribute addProperty Id "InputAT %I*ARRAY[0..7] OF BOOL8Sync_ErrorAT %I*BOOL1"}
{attribute addProperty CRC "2788215981"}
{attribute addProperty Size "9"}
TYPE DO_Diag_Inputs_CC455148 EXTENDS InputBase_8311D824 :
STRUCT
	{attribute addProperty Name "Input"}
	Input AT %I* : ARRAY[0..7] OF BOOL;
	{attribute addProperty Name "Sync_Error"}
	Sync_Error AT %I* : BOOL;
END_STRUCT
END_TYPE

// ---- DUTs/IO/PDOs/DO_Diag_Inputs_212B82C1.TcDUT
{attribute 'GeneratedUsingTerminal: EP2316-0008-0017'}
{attribute addProperty BoxType "EP2316-0008-0017"}
{attribute addProperty Id "Diag_InputAT %I*ARRAY[0..7] OF BOOL8Sync_ErrorAT %I*BOOL1"}
{attribute addProperty CRC "3811544510"}
{attribute addProperty Size "9"}
TYPE DO_Diag_Inputs_212B82C1 EXTENDS InputBase_8311D824 :
STRUCT
	{attribute addProperty Name "Diag_Input"}
	Diag_Input AT %I* : ARRAY[0..7] OF BOOL;
	{attribute addProperty Name "Sync_Error"}
	Sync_Error AT %I* : BOOL;
END_STRUCT
END_TYPE

// ---- DUTs/IO/PDOs/DO_Inputs_Device_AF161A9E.TcDUT
{attribute 'GeneratedUsingTerminal: EP2316-0008-0017'}
{attribute addProperty BoxType "EP2316-0008-0017"}
{attribute addProperty Id "Safe_state_activeAT %I*BOOL1Error_channel_1AT %I*BOOL1Sync_ErrorAT %I*BOOL1TxPDO_ToggleAT %I*BOOL1"}
{attribute addProperty CRC "2937461406"}
{attribute addProperty Size "4"}
TYPE DO_Inputs_Device_AF161A9E EXTENDS InputBase_8311D824 :
STRUCT
	{attribute addProperty Name "Safe_state_active"}
	Safe_state_active AT %I* : BOOL;
	{attribute addProperty Name "Error_channel_1"}
	Error_channel_1 AT %I* : BOOL;
	{attribute addProperty Name "Sync_Error"}
	Sync_Error AT %I* : BOOL;
	{attribute addProperty Name "TxPDO_Toggle"}
	TxPDO_Toggle AT %I* : BOOL;
END_STRUCT
END_TYPE

// ---- DUTs/IO/PDOs/DO_Outputs_28AC1A9E.TcDUT
{attribute 'GeneratedUsingTerminal: EP2316-0008-0017'}
{attribute addProperty BoxType "EP2316-0008-0017"}
{attribute addProperty Id "OutputAT %Q*ARRAY[0..7] OF BOOL8"}
{attribute addProperty CRC "1253840710"}
{attribute addProperty Size "8"}
TYPE DO_Outputs_28AC1A9E EXTENDS OutputBase_10CEE7DE :
STRUCT
	{attribute addProperty Name "Output"}
	Output AT %Q* : ARRAY[0..7] OF BOOL;
END_STRUCT
END_TYPE

// ---- DUTs/IO/PDOs/DO_Outputs_Device_36A5EF17.TcDUT
{attribute 'GeneratedUsingTerminal: EP2316-0008-0017'}
{attribute addProperty BoxType "EP2316-0008-0017"}
{attribute addProperty Id "Set_safe_stateAT %Q*BOOL1Reset_outputsAT %Q*BOOL1"}
{attribute addProperty CRC "916844311"}
{attribute addProperty Size "2"}
TYPE DO_Outputs_Device_36A5EF17 EXTENDS OutputBase_10CEE7DE :
STRUCT
	{attribute addProperty Name "Set_safe_state"}
	Set_safe_state AT %Q* : BOOL;
	{attribute addProperty Name "Reset_outputs"}
	Reset_outputs AT %Q* : BOOL;
END_STRUCT
END_TYPE

// ---- DUTs/IO/PDOs/InfoData_32EB74EA.TcDUT
{attribute 'GeneratedUsingTerminal: EP2316-0008-0017'}
{attribute addProperty BoxType "EP2316-0008-0017"}
{attribute addProperty Id "AdsAddrAT %I*AMSADDR8StateAT %I*UINT2"}
{attribute addProperty CRC "854291690"}
{attribute addProperty Size "10"}
TYPE InfoData_32EB74EA EXTENDS InputBase_8311D824 :
STRUCT
	{attribute addProperty Name "AdsAddr"}
	AdsAddr AT %I* : AMSADDR;
	{attribute addProperty Name "State"}
	State AT %I* : UINT;
END_STRUCT
END_TYPE

// ---- DUTs/IO/PDOs/InfoData_0A66F009.TcDUT
{attribute 'GeneratedUsingTerminal: EP2339-0021-0016'}
{attribute addProperty BoxType "EP2339-0021-0016"}
{attribute addProperty Id "AoeNetIdAT %I*AMSNETID6StateAT %I*UINT2"}
{attribute addProperty CRC "174518281"}
{attribute addProperty Size "8"}
TYPE InfoData_0A66F009 EXTENDS InputBase_8311D824 :
STRUCT
	{attribute addProperty Name "AoeNetId"}
	AoeNetId AT %I* : AMSNETID;
	{attribute addProperty Name "State"}
	State AT %I* : UINT;
END_STRUCT
END_TYPE

// ---- DUTs/IO/PDOs/ENC_Inputs_B3536485.TcDUT
{attribute 'GeneratedUsingTerminal: EJ5151-0000-0016'}
{attribute addProperty BoxType "EJ5151-0000-0016"}
{attribute addProperty Id "StatusAT %I*Status_3E6F3FF310Counter_valueAT %I*UINT2Latch_valueAT %I*UINT2"}
{attribute addProperty CRC "3008586885"}
{attribute addProperty Size "14"}
TYPE ENC_Inputs_B3536485 EXTENDS InputBase_8311D824 :
STRUCT
	{attribute addProperty Name "Status"}
	Status AT %I* : Status_3E6F3FF3;
	{attribute addProperty Name "Counter_value"}
	Counter_value AT %I* : UINT;
	{attribute addProperty Name "Latch_value"}
	Latch_value AT %I* : UINT;
END_STRUCT
END_TYPE

// ---- DUTs/IO/PDOs/ENC_Inputs_24B63C53.TcDUT
{attribute 'GeneratedUsingTerminal: EJ5151-0000-0016'}
{attribute addProperty BoxType "EJ5151-0000-0016"}
{attribute addProperty Id "Period_valueAT %I*UDINT4"}
{attribute addProperty CRC "615922771"}
{attribute addProperty Size "4"}
TYPE ENC_Inputs_24B63C53 EXTENDS InputBase_8311D824 :
STRUCT
	{attribute addProperty Name "Period_value"}
	Period_value AT %I* : UDINT;
END_STRUCT
END_TYPE

// ---- DUTs/IO/PDOs/ENC_Outputs_21E2D14D.TcDUT
{attribute 'GeneratedUsingTerminal: EJ5151-0000-0016'}
{attribute addProperty BoxType "EJ5151-0000-0016"}
{attribute addProperty Id "ControlAT %Q*Control_6EF2C5D04Set_counter_valueAT %Q*UINT2"}
{attribute addProperty CRC "568512845"}
{attribute addProperty Size "6"}
TYPE ENC_Outputs_21E2D14D EXTENDS OutputBase_10CEE7DE :
STRUCT
	{attribute addProperty Name "Control"}
	Control AT %Q* : Control_6EF2C5D0;
	{attribute addProperty Name "Set_counter_value"}
	Set_counter_value AT %Q* : UINT;
END_STRUCT
END_TYPE

// ---- DUTs/IO/PDOs/Ch1_CycleCount_9DBE2BC5.TcDUT
{attribute 'GeneratedUsingTerminal: EL1262-0000-0002'}
{attribute addProperty BoxType "EL1262-0000-0002"}
{attribute addProperty Id "Ch1_CycleCountAT %I*UINT2"}
{attribute addProperty CRC "2646485957"}
{attribute addProperty Size "2"}
TYPE Ch1_CycleCount_9DBE2BC5 EXTENDS InputBase_8311D824 :
STRUCT
	{attribute addProperty Name "Ch1_CycleCount"}
	Ch1_CycleCount AT %I* : UINT;
END_STRUCT
END_TYPE

// ---- DUTs/IO/PDOs/Ch1_Input_FFC4CE24.TcDUT
{attribute 'GeneratedUsingTerminal: EL1262-0000-0002'}
{attribute addProperty BoxType "EL1262-0000-0002"}
{attribute addProperty Id "Ch1_InputAT %I*BOOL1"}
{attribute addProperty CRC "4291087908"}
{attribute addProperty Size "1"}
TYPE Ch1_Input_FFC4CE24 EXTENDS InputBase_8311D824 :
STRUCT
	{attribute addProperty Name "Ch1_Input"}
	Ch1_Input AT %I* : BOOL;
END_STRUCT
END_TYPE

// ---- DUTs/IO/PDOs/EMPTY_STRUCTURE.TcDUT
{attribute 'GeneratedUsingTerminal: EL1262-0000-0002'}
{attribute addProperty BoxType "EL1262-0000-0002"}
{attribute addProperty Id "EMPTY_STRUCTURE"}
{attribute addProperty CRC "0"}
{attribute addProperty Size "0"}
TYPE EMPTY_STRUCTURE :
STRUCT
END_STRUCT
END_TYPE

// ---- DUTs/IO/PDOs/Ch2_CycleCount_976A51B5.TcDUT
{attribute 'GeneratedUsingTerminal: EL1262-0000-0002'}
{attribute addProperty BoxType "EL1262-0000-0002"}
{attribute addProperty Id "Ch2_CycleCountAT %I*UINT2"}
{attribute addProperty CRC "2540327349"}
{attribute addProperty Size "2"}
TYPE Ch2_CycleCount_976A51B5 EXTENDS InputBase_8311D824 :
STRUCT
	{attribute addProperty Name "Ch2_CycleCount"}
	Ch2_CycleCount AT %I* : UINT;
END_STRUCT
END_TYPE

// ---- DUTs/IO/PDOs/Ch2_Input_78ADA90C.TcDUT
{attribute 'GeneratedUsingTerminal: EL1262-0000-0002'}
{attribute addProperty BoxType "EL1262-0000-0002"}
{attribute addProperty Id "Ch2_InputAT %I*BOOL1"}
{attribute addProperty CRC "2024646924"}
{attribute addProperty Size "1"}
TYPE Ch2_Input_78ADA90C EXTENDS InputBase_8311D824 :
STRUCT
	{attribute addProperty Name "Ch2_Input"}
	Ch2_Input AT %I* : BOOL;
END_STRUCT
END_TYPE

// ---- DUTs/IO/PDOs/NextSync1Time_EE185E17.TcDUT
{attribute 'GeneratedUsingTerminal: EL1262-0000-0002'}
{attribute addProperty BoxType "EL1262-0000-0002"}
{attribute addProperty Id "StartTimeNextLatchAT %I*UDINT4"}
{attribute addProperty CRC "3994574359"}
{attribute addProperty Size "4"}
TYPE NextSync1Time_EE185E17 EXTENDS InputBase_8311D824 :
STRUCT
	{attribute addProperty Name "StartTimeNextLatch"}
	StartTimeNextLatch AT %I* : UDINT;
END_STRUCT
END_TYPE

// ---- DUTs/IO/PDOs/InfoData_A7436BC6.TcDUT
{attribute 'GeneratedUsingTerminal: EL1262-0000-0002'}
{attribute addProperty BoxType "EL1262-0000-0002"}
{attribute addProperty Id "DcOutputShiftAT %I*DINT4DcInputShiftAT %I*DINT4StateAT %I*UINT2"}
{attribute addProperty CRC "2806213574"}
{attribute addProperty Size "10"}
TYPE InfoData_A7436BC6 EXTENDS InputBase_8311D824 :
STRUCT
	{attribute addProperty Name "DcOutputShift"}
	DcOutputShift AT %I* : DINT;
	{attribute addProperty Name "DcInputShift"}
	DcInputShift AT %I* : DINT;
	{attribute addProperty Name "State"}
	State AT %I* : UINT;
END_STRUCT
END_TYPE

// ---- DUTs/IO/PDOs/CycCount0_2C233804.TcDUT
{attribute 'GeneratedUsingTerminal: EL2262-0000-0001'}
{attribute addProperty BoxType "EL2262-0000-0001"}
{attribute addProperty Id "Cycle_CounterAT %Q*UINT2"}
{attribute addProperty CRC "740505604"}
{attribute addProperty Size "2"}
TYPE CycCount0_2C233804 EXTENDS OutputBase_10CEE7DE :
STRUCT
	{attribute addProperty Name "Cycle_Counter"}
	Cycle_Counter AT %Q* : UINT;
END_STRUCT
END_TYPE

// ---- DUTs/IO/PDOs/Sample_0023574C.TcDUT
{attribute 'GeneratedUsingTerminal: EL2262-0000-0001'}
{attribute addProperty BoxType "EL2262-0000-0001"}
{attribute addProperty Id "Output0AT %Q*BOOL1"}
{attribute addProperty CRC "2316108"}
{attribute addProperty Size "1"}
TYPE Sample_0023574C EXTENDS OutputBase_10CEE7DE :
STRUCT
	{attribute addProperty Name "Output0"}
	Output0 AT %Q* : BOOL;
END_STRUCT
END_TYPE

// ---- DUTs/IO/PDOs/CycCount1_2C233804.TcDUT
{attribute 'GeneratedUsingTerminal: EL2262-0000-0001'}
{attribute addProperty BoxType "EL2262-0000-0001"}
{attribute addProperty Id "Cycle_CounterAT %Q*UINT2"}
{attribute addProperty CRC "740505604"}
{attribute addProperty Size "2"}
TYPE CycCount1_2C233804 EXTENDS OutputBase_10CEE7DE :
STRUCT
	{attribute addProperty Name "Cycle_Counter"}
	Cycle_Counter AT %Q* : UINT;
END_STRUCT
END_TYPE

// ---- DUTs/IO/PDOs/Sample_07D5B44A.TcDUT
{attribute 'GeneratedUsingTerminal: EL2262-0000-0001'}
{attribute addProperty BoxType "EL2262-0000-0001"}
{attribute addProperty Id "Output1AT %Q*BOOL1"}
{attribute addProperty CRC "131445834"}
{attribute addProperty Size "1"}
TYPE Sample_07D5B44A EXTENDS OutputBase_10CEE7DE :
STRUCT
	{attribute addProperty Name "Output1"}
	Output1 AT %Q* : BOOL;
END_STRUCT
END_TYPE

// ---- DUTs/IO/PDOs/WcState_0B2B16F9.TcDUT
{attribute 'GeneratedUsingTerminal: EL2262-0000-0001'}
{attribute addProperty BoxType "EL2262-0000-0001"}
{attribute addProperty Id "WcStateAT %I*BOOL1"}
{attribute addProperty CRC "187373305"}
{attribute addProperty Size "1"}
TYPE WcState_0B2B16F9 :
STRUCT
	{attribute addProperty Name "WcState"}
	WcState AT %I* : BOOL;
END_STRUCT
END_TYPE

// ---- DUTs/IO/PDOs/CycCount0_AF431CE0.TcDUT
{attribute 'GeneratedUsingTerminal: EL2262-0000-0002'}
{attribute addProperty BoxType "EL2262-0000-0002"}
{attribute addProperty Id "Cycle_Counter0AT %Q*UINT2"}
{attribute addProperty CRC "2940411104"}
{attribute addProperty Size "2"}
TYPE CycCount0_AF431CE0 EXTENDS OutputBase_10CEE7DE :
STRUCT
	{attribute addProperty Name "Cycle_Counter0"}
	Cycle_Counter0 AT %Q* : UINT;
END_STRUCT
END_TYPE

// ---- DUTs/IO/PDOs/CycCount1_A8B5FFE6.TcDUT
{attribute 'GeneratedUsingTerminal: EL2262-0000-0002'}
{attribute addProperty BoxType "EL2262-0000-0002"}
{attribute addProperty Id "Cycle_Counter1AT %Q*UINT2"}
{attribute addProperty CRC "2830499814"}
{attribute addProperty Size "2"}
TYPE CycCount1_A8B5FFE6 EXTENDS OutputBase_10CEE7DE :
STRUCT
	{attribute addProperty Name "Cycle_Counter1"}
	Cycle_Counter1 AT %Q* : UINT;
END_STRUCT
END_TYPE

// ---- DUTs/IO/PDOs/StartTimeNextOutput_228767F4.TcDUT
{attribute 'GeneratedUsingTerminal: EL2262-0000-0004'}
{attribute addProperty BoxType "EL2262-0000-0004"}
{attribute addProperty Id "StartTimeNextOutputAT %I*UDINT4"}
{attribute addProperty CRC "579299316"}
{attribute addProperty Size "4"}
TYPE StartTimeNextOutput_228767F4 EXTENDS InputBase_8311D824 :
STRUCT
	{attribute addProperty Name "StartTimeNextOutput"}
	StartTimeNextOutput AT %I* : UDINT;
END_STRUCT
END_TYPE

// ---- DUTs/IO/PDOs/SAI_Inputs_3A838E11.TcDUT
{attribute 'GeneratedUsingTerminal: EL3681-0000-0017'}
{attribute addProperty BoxType "EL3681-0000-0017"}
{attribute addProperty Id "StatusAT %I*Status_237FCB0F10ValueAT %I*DINT4"}
{attribute addProperty CRC "981700113"}
{attribute addProperty Size "14"}
TYPE SAI_Inputs_3A838E11 EXTENDS InputBase_8311D824 :
STRUCT
	{attribute addProperty Name "Status"}
	Status AT %I* : Status_237FCB0F;
	{attribute addProperty Name "Value"}
	Value AT %I* : DINT;
END_STRUCT
END_TYPE

// ---- DUTs/IO/PDOs/SAI_Range_C3200E78.TcDUT
{attribute 'GeneratedUsingTerminal: EL3681-0000-0017'}
{attribute addProperty BoxType "EL3681-0000-0017"}
{attribute addProperty Id "SettingAT %I*Setting_24C049402"}
{attribute addProperty CRC "3273657976"}
{attribute addProperty Size "2"}
TYPE SAI_Range_C3200E78 EXTENDS InputBase_8311D824 :
STRUCT
	{attribute addProperty Name "Setting"}
	Setting AT %I* : Setting_24C04940;
END_STRUCT
END_TYPE

// ---- DUTs/IO/PDOs/SAI_Range_3710D747.TcDUT
{attribute 'GeneratedUsingTerminal: EL3681-0000-0017'}
{attribute addProperty BoxType "EL3681-0000-0017"}
{attribute addProperty Id "CtrlAT %Q*Ctrl_56BB2DF23"}
{attribute addProperty CRC "923850567"}
{attribute addProperty Size "3"}
TYPE SAI_Range_3710D747 EXTENDS OutputBase_10CEE7DE :
STRUCT
	{attribute addProperty Name "Ctrl"}
	Ctrl AT %Q* : Ctrl_56BB2DF2;
END_STRUCT
END_TYPE

// ---- DUTs/IO/PDOs/SAI_Inputs_84B29FE9.TcDUT
{attribute 'GeneratedUsingTerminal: EL3681-0000-0018'}
{attribute addProperty BoxType "EL3681-0000-0018"}
{attribute addProperty Id "StatusAT %I*Status_51F0A92410ValueAT %I*DINT4"}
{attribute addProperty CRC "2226298857"}
{attribute addProperty Size "14"}
TYPE SAI_Inputs_84B29FE9 EXTENDS InputBase_8311D824 :
STRUCT
	{attribute addProperty Name "Status"}
	Status AT %I* : Status_51F0A924;
	{attribute addProperty Name "Value"}
	Value AT %I* : DINT;
END_STRUCT
END_TYPE

// ---- DUTs/IO/PDOs/SAI_Range_BDBF6DA9.TcDUT
{attribute 'GeneratedUsingTerminal: EL3681-0000-0018'}
{attribute addProperty BoxType "EL3681-0000-0018"}
{attribute addProperty Id "SettingsAT %I*Settings_24C049402"}
{attribute addProperty CRC "3183439273"}
{attribute addProperty Size "2"}
TYPE SAI_Range_BDBF6DA9 EXTENDS InputBase_8311D824 :
STRUCT
	{attribute addProperty Name "Settings"}
	Settings AT %I* : Settings_24C04940;
END_STRUCT
END_TYPE

// ---- DUTs/IO/PDOs/SAI_Range_2A187FC5.TcDUT
{attribute 'GeneratedUsingTerminal: EL3681-0000-0018'}
{attribute addProperty BoxType "EL3681-0000-0018"}
{attribute addProperty Id "ControlAT %Q*Control_18D542D94"}
{attribute addProperty CRC "706248645"}
{attribute addProperty Size "4"}
TYPE SAI_Range_2A187FC5 EXTENDS OutputBase_10CEE7DE :
STRUCT
	{attribute addProperty Name "Control"}
	Control AT %Q* : Control_18D542D9;
END_STRUCT
END_TYPE

// ---- DUTs/IO/PDOs/Channel_B90637B9.TcDUT
{attribute 'GeneratedUsingTerminal: EL5101--0000'}
{attribute addProperty BoxType "EL5101--0000"}
{attribute addProperty Id "StatusAT %I*USINT1ValueAT %I*UINT2LatchAT %I*UINT2"}
{attribute addProperty CRC "3104192441"}
{attribute addProperty Size "5"}
TYPE Channel_B90637B9 EXTENDS InputBase_8311D824 :
STRUCT
	{attribute addProperty Name "Status"}
	Status AT %I* : USINT;
	{attribute addProperty Name "Value"}
	Value AT %I* : UINT;
	{attribute addProperty Name "Latch"}
	Latch AT %I* : UINT;
END_STRUCT
END_TYPE

// ---- DUTs/IO/PDOs/Channel_C6781B15.TcDUT
{attribute 'GeneratedUsingTerminal: EL5101--0000'}
{attribute addProperty BoxType "EL5101--0000"}
{attribute addProperty Id "CtrlAT %Q*USINT1ValueAT %Q*UINT2"}
{attribute addProperty CRC "3329760021"}
{attribute addProperty Size "3"}
TYPE Channel_C6781B15 EXTENDS OutputBase_10CEE7DE :
STRUCT
	{attribute addProperty Name "Ctrl"}
	Ctrl AT %Q* : USINT;
	{attribute addProperty Name "Value"}
	Value AT %Q* : UINT;
END_STRUCT
END_TYPE

// ---- DUTs/IO/PDOs/ENC_Inputs_3399C5AA.TcDUT
{attribute 'GeneratedUsingTerminal: EL5151-0000-0016'}
{attribute addProperty BoxType "EL5151-0000-0016"}
{attribute addProperty Id "StatusAT %I*Status_396FCBA08Counter_valueAT %I*UDINT4Latch_valueAT %I*UDINT4"}
{attribute addProperty CRC "865715626"}
{attribute addProperty Size "16"}
TYPE ENC_Inputs_3399C5AA EXTENDS InputBase_8311D824 :
STRUCT
	{attribute addProperty Name "Status"}
	Status AT %I* : Status_396FCBA0;
	{attribute addProperty Name "Counter_value"}
	Counter_value AT %I* : UDINT;
	{attribute addProperty Name "Latch_value"}
	Latch_value AT %I* : UDINT;
END_STRUCT
END_TYPE

// ---- DUTs/IO/PDOs/ENC_Outputs_2E45048F.TcDUT
{attribute 'GeneratedUsingTerminal: EL5151-0000-0016'}
{attribute addProperty BoxType "EL5151-0000-0016"}
{attribute addProperty Id "Enable_latch_CAT %Q*BOOL1Enable_latch_extern_on_positive_edgeAT %Q*BOOL1Set_counterAT %Q*BOOL1Enable_latch_extern_on_negative_edgeAT %Q*BOOL1Set_counter_valueAT %Q*UDINT4"}
{attribute addProperty CRC "776275087"}
{attribute addProperty Size "8"}
TYPE ENC_Outputs_2E45048F EXTENDS OutputBase_10CEE7DE :
STRUCT
	{attribute addProperty Name "Enable_latch_C"}
	Enable_latch_C AT %Q* : BOOL;
	{attribute addProperty Name "Enable_latch_extern_on_positive_edge"}
	Enable_latch_extern_on_positive_edge AT %Q* : BOOL;
	{attribute addProperty Name "Set_counter"}
	Set_counter AT %Q* : BOOL;
	{attribute addProperty Name "Enable_latch_extern_on_negative_edge"}
	Enable_latch_extern_on_negative_edge AT %Q* : BOOL;
	{attribute addProperty Name "Set_counter_value"}
	Set_counter_value AT %Q* : UDINT;
END_STRUCT
END_TYPE

// ---- DUTs/IO/PDOs/ENC_Inputs_561E041F.TcDUT
{attribute 'GeneratedUsingTerminal: EL5151-0000-0017'}
{attribute addProperty BoxType "EL5151-0000-0017"}
{attribute addProperty Id "Latch_C_validAT %I*BOOL1Latch_extern_validAT %I*BOOL1Set_counter_doneAT %I*BOOL1Extrapolation_stallAT %I*BOOL1Status_of_input_AAT %I*BOOL1Status_of_input_BAT %I*BOOL1Status_of_input_CAT %I*BOOL1Status_of_extern_latchAT %I*BOOL1Sync_ErrorAT %I*BOOL1TxPDO_ToggleAT %I*BOOL1Counter_valueAT %I*UDINT4Latch_valueAT %I*UDINT4"}
{attribute addProperty CRC "1444807711"}
{attribute addProperty Size "18"}
TYPE ENC_Inputs_561E041F EXTENDS InputBase_8311D824 :
STRUCT
	{attribute addProperty Name "Latch_C_valid"}
	Latch_C_valid AT %I* : BOOL;
	{attribute addProperty Name "Latch_extern_valid"}
	Latch_extern_valid AT %I* : BOOL;
	{attribute addProperty Name "Set_counter_done"}
	Set_counter_done AT %I* : BOOL;
	{attribute addProperty Name "Extrapolation_stall"}
	Extrapolation_stall AT %I* : BOOL;
	{attribute addProperty Name "Status_of_input_A"}
	Status_of_input_A AT %I* : BOOL;
	{attribute addProperty Name "Status_of_input_B"}
	Status_of_input_B AT %I* : BOOL;
	{attribute addProperty Name "Status_of_input_C"}
	Status_of_input_C AT %I* : BOOL;
	{attribute addProperty Name "Status_of_extern_latch"}
	Status_of_extern_latch AT %I* : BOOL;
	{attribute addProperty Name "Sync_Error"}
	Sync_Error AT %I* : BOOL;
	{attribute addProperty Name "TxPDO_Toggle"}
	TxPDO_Toggle AT %I* : BOOL;
	{attribute addProperty Name "Counter_value"}
	Counter_value AT %I* : UDINT;
	{attribute addProperty Name "Latch_value"}
	Latch_value AT %I* : UDINT;
END_STRUCT
END_TYPE

// ---- DUTs/IO/PDOs/ENC_Inputs_F139456B.TcDUT
{attribute 'GeneratedUsingTerminal: EL5151-0080-0016'}
{attribute addProperty BoxType "EL5151-0080-0016"}
{attribute addProperty Id "Latch_C_validAT %I*BOOL1Latch_extern_validAT %I*BOOL1Set_counter_doneAT %I*BOOL1Extrapolation_stallAT %I*BOOL1Status_of_input_AAT %I*BOOL1Status_of_input_BAT %I*BOOL1Status_of_input_CAT %I*BOOL1Status_of_extern_latchAT %I*BOOL1Sync_ErrorAT %I*BOOL1TxPDO_ToggleAT %I*BOOL1Counter_valueAT %I*UINT2Latch_valueAT %I*UINT2"}
{attribute addProperty CRC "4047062379"}
{attribute addProperty Size "14"}
TYPE ENC_Inputs_F139456B EXTENDS InputBase_8311D824 :
STRUCT
	{attribute addProperty Name "Latch_C_valid"}
	Latch_C_valid AT %I* : BOOL;
	{attribute addProperty Name "Latch_extern_valid"}
	Latch_extern_valid AT %I* : BOOL;
	{attribute addProperty Name "Set_counter_done"}
	Set_counter_done AT %I* : BOOL;
	{attribute addProperty Name "Extrapolation_stall"}
	Extrapolation_stall AT %I* : BOOL;
	{attribute addProperty Name "Status_of_input_A"}
	Status_of_input_A AT %I* : BOOL;
	{attribute addProperty Name "Status_of_input_B"}
	Status_of_input_B AT %I* : BOOL;
	{attribute addProperty Name "Status_of_input_C"}
	Status_of_input_C AT %I* : BOOL;
	{attribute addProperty Name "Status_of_extern_latch"}
	Status_of_extern_latch AT %I* : BOOL;
	{attribute addProperty Name "Sync_Error"}
	Sync_Error AT %I* : BOOL;
	{attribute addProperty Name "TxPDO_Toggle"}
	TxPDO_Toggle AT %I* : BOOL;
	{attribute addProperty Name "Counter_value"}
	Counter_value AT %I* : UINT;
	{attribute addProperty Name "Latch_value"}
	Latch_value AT %I* : UINT;
END_STRUCT
END_TYPE

// ---- DUTs/IO/PDOs/ENC_Outputs_6FDDC669.TcDUT
{attribute 'GeneratedUsingTerminal: EL5151-0080-0016'}
{attribute addProperty BoxType "EL5151-0080-0016"}
{attribute addProperty Id "Enable_latch_CAT %Q*BOOL1Enable_latch_extern_on_positive_edgeAT %Q*BOOL1Set_counterAT %Q*BOOL1Enable_latch_extern_on_negative_edgeAT %Q*BOOL1Set_counter_valueAT %Q*UINT2"}
{attribute addProperty CRC "1876805225"}
{attribute addProperty Size "6"}
TYPE ENC_Outputs_6FDDC669 EXTENDS OutputBase_10CEE7DE :
STRUCT
	{attribute addProperty Name "Enable_latch_C"}
	Enable_latch_C AT %Q* : BOOL;
	{attribute addProperty Name "Enable_latch_extern_on_positive_edge"}
	Enable_latch_extern_on_positive_edge AT %Q* : BOOL;
	{attribute addProperty Name "Set_counter"}
	Set_counter AT %Q* : BOOL;
	{attribute addProperty Name "Enable_latch_extern_on_negative_edge"}
	Enable_latch_extern_on_negative_edge AT %Q* : BOOL;
	{attribute addProperty Name "Set_counter_value"}
	Set_counter_value AT %Q* : UINT;
END_STRUCT
END_TYPE

// ---- DUTs/IO/PDOs/L1_Voltage_Status_784F03AD.TcDUT
{attribute 'GeneratedUsingTerminal: EL3773-0000-0016'}
{attribute addProperty BoxType "EL3773-0000-0016"}
{attribute addProperty Id "U1_STATUSAT %I*U1_STATUS_B07533568"}
{attribute addProperty CRC "2018444205"}
{attribute addProperty Size "8"}
TYPE L1_Voltage_Status_784F03AD EXTENDS InputBase_8311D824 :
STRUCT
	{attribute addProperty Name "U1_STATUS"}
	U1_STATUS AT %I* : U1_STATUS_B0753356;
END_STRUCT
END_TYPE

// ---- DUTs/IO/PDOs/L1_Voltage_Samples_ED678DEE.TcDUT
{attribute 'GeneratedUsingTerminal: EL3773-0000-0016'}
{attribute addProperty BoxType "EL3773-0000-0016"}
{attribute addProperty Id "U1_SAMPLESAT %I*U1_SAMPLES_2D13B74B20"}
{attribute addProperty CRC "3982986734"}
{attribute addProperty Size "20"}
TYPE L1_Voltage_Samples_ED678DEE EXTENDS InputBase_8311D824 :
STRUCT
	{attribute addProperty Name "U1_SAMPLES"}
	U1_SAMPLES AT %I* : U1_SAMPLES_2D13B74B;
END_STRUCT
END_TYPE

// ---- DUTs/IO/PDOs/L1_Current_Samples_89E07818.TcDUT
{attribute 'GeneratedUsingTerminal: EL3773-0000-0016'}
{attribute addProperty BoxType "EL3773-0000-0016"}
{attribute addProperty Id "I1_STATUSAT %I*I1_STATUS_B07533568"}
{attribute addProperty CRC "2313189400"}
{attribute addProperty Size "8"}
TYPE L1_Current_Samples_89E07818 EXTENDS InputBase_8311D824 :
STRUCT
	{attribute addProperty Name "I1_STATUS"}
	I1_STATUS AT %I* : I1_STATUS_B0753356;
END_STRUCT
END_TYPE

// ---- DUTs/IO/PDOs/L1_Current_Samples_3209B12F.TcDUT
{attribute 'GeneratedUsingTerminal: EL3773-0000-0016'}
{attribute addProperty BoxType "EL3773-0000-0016"}
{attribute addProperty Id "I1_SAMPLESAT %I*I1_SAMPLES_2D13B74B20"}
{attribute addProperty CRC "839495983"}
{attribute addProperty Size "20"}
TYPE L1_Current_Samples_3209B12F EXTENDS InputBase_8311D824 :
STRUCT
	{attribute addProperty Name "I1_SAMPLES"}
	I1_SAMPLES AT %I* : I1_SAMPLES_2D13B74B;
END_STRUCT
END_TYPE

// ---- DUTs/IO/PDOs/L2_Voltage_Status_0626A010.TcDUT
{attribute 'GeneratedUsingTerminal: EL3773-0000-0016'}
{attribute addProperty BoxType "EL3773-0000-0016"}
{attribute addProperty Id "U2_STATUSAT %I*U2_STATUS_B07533568"}
{attribute addProperty CRC "103194640"}
{attribute addProperty Size "8"}
TYPE L2_Voltage_Status_0626A010 EXTENDS InputBase_8311D824 :
STRUCT
	{attribute addProperty Name "U2_STATUS"}
	U2_STATUS AT %I* : U2_STATUS_B0753356;
END_STRUCT
END_TYPE

// ---- DUTs/IO/PDOs/L2_Voltage_Samples_D91109BE.TcDUT
{attribute 'GeneratedUsingTerminal: EL3773-0000-0016'}
{attribute addProperty BoxType "EL3773-0000-0016"}
{attribute addProperty Id "U2_SAMPLESAT %I*U2_SAMPLES_2D13B74B20"}
{attribute addProperty CRC "3641772478"}
{attribute addProperty Size "20"}
TYPE L2_Voltage_Samples_D91109BE EXTENDS InputBase_8311D824 :
STRUCT
	{attribute addProperty Name "U2_SAMPLES"}
	U2_SAMPLES AT %I* : U2_SAMPLES_2D13B74B;
END_STRUCT
END_TYPE

// ---- DUTs/IO/PDOs/L2_Current_Status_F789DBA5.TcDUT
{attribute 'GeneratedUsingTerminal: EL3773-0000-0016'}
{attribute addProperty BoxType "EL3773-0000-0016"}
{attribute addProperty Id "I2_STATUSAT %I*I2_STATUS_B07533568"}
{attribute addProperty CRC "4153007013"}
{attribute addProperty Size "8"}
TYPE L2_Current_Status_F789DBA5 EXTENDS InputBase_8311D824 :
STRUCT
	{attribute addProperty Name "I2_STATUS"}
	I2_STATUS AT %I* : I2_STATUS_B0753356;
END_STRUCT
END_TYPE

// ---- DUTs/IO/PDOs/L2_Current_Samples_067F357F.TcDUT
{attribute 'GeneratedUsingTerminal: EL3773-0000-0016'}
{attribute addProperty BoxType "EL3773-0000-0016"}
{attribute addProperty Id "I2_SAMPLESAT %I*I2_SAMPLES_2D13B74B20"}
{attribute addProperty CRC "109000063"}
{attribute addProperty Size "20"}
TYPE L2_Current_Samples_067F357F EXTENDS InputBase_8311D824 :
STRUCT
	{attribute addProperty Name "I2_SAMPLES"}
	I2_SAMPLES AT %I* : I2_SAMPLES_2D13B74B;
END_STRUCT
END_TYPE

// ---- DUTs/IO/PDOs/L3_Voltage_Status_2C01C17B.TcDUT
{attribute 'GeneratedUsingTerminal: EL3773-0000-0016'}
{attribute addProperty BoxType "EL3773-0000-0016"}
{attribute addProperty Id "U3_STATUSAT %I*U3_STATUS_B07533568"}
{attribute addProperty CRC "738312571"}
{attribute addProperty Size "8"}
TYPE L3_Voltage_Status_2C01C17B EXTENDS InputBase_8311D824 :
STRUCT
	{attribute addProperty Name "U3_STATUS"}
	U3_STATUS AT %I* : U3_STATUS_B0753356;
END_STRUCT
END_TYPE

// ---- DUTs/IO/PDOs/L3_Voltage_Samples_CAC3758E.TcDUT
{attribute 'GeneratedUsingTerminal: EL3773-0000-0016'}
{attribute addProperty BoxType "EL3773-0000-0016"}
{attribute addProperty Id "U3_SAMPLESAT %I*U3_SAMPLES_2D13B74B20"}
{attribute addProperty CRC "3401807246"}
{attribute addProperty Size "20"}
TYPE L3_Voltage_Samples_CAC3758E EXTENDS InputBase_8311D824 :
STRUCT
	{attribute addProperty Name "U3_SAMPLES"}
	U3_SAMPLES AT %I* : U3_SAMPLES_2D13B74B;
END_STRUCT
END_TYPE

// ---- DUTs/IO/PDOs/L3_Current_Status_DDAEBACE.TcDUT
{attribute 'GeneratedUsingTerminal: EL3773-0000-0016'}
{attribute addProperty BoxType "EL3773-0000-0016"}
{attribute addProperty Id "I3_STATUSAT %I*I3_STATUS_B07533568"}
{attribute addProperty CRC "3719215822"}
{attribute addProperty Size "8"}
TYPE L3_Current_Status_DDAEBACE EXTENDS InputBase_8311D824 :
STRUCT
	{attribute addProperty Name "I3_STATUS"}
	I3_STATUS AT %I* : I3_STATUS_B0753356;
END_STRUCT
END_TYPE

// ---- DUTs/IO/PDOs/L3_Current_Samples_15AD494F.TcDUT
{attribute 'GeneratedUsingTerminal: EL3773-0000-0016'}
{attribute addProperty BoxType "EL3773-0000-0016"}
{attribute addProperty Id "I3_SAMPLESAT %I*I3_SAMPLES_2D13B74B20"}
{attribute addProperty CRC "363678031"}
{attribute addProperty Size "20"}
TYPE L3_Current_Samples_15AD494F EXTENDS InputBase_8311D824 :
STRUCT
	{attribute addProperty Name "I3_SAMPLES"}
	I3_SAMPLES AT %I* : I3_SAMPLES_2D13B74B;
END_STRUCT
END_TYPE

// ---- DUTs/IO/PDOs/AI_Timestamp_NextSync1Time_9AFDC275.TcDUT
{attribute 'GeneratedUsingTerminal: EL3773-0000-0016'}
{attribute addProperty BoxType "EL3773-0000-0016"}
{attribute addProperty Id "StartTimeNextLatchAT %I*ULINT8"}
{attribute addProperty CRC "2600321653"}
{attribute addProperty Size "8"}
TYPE AI_Timestamp_NextSync1Time_9AFDC275 EXTENDS InputBase_8311D824 :
STRUCT
	{attribute addProperty Name "StartTimeNextLatch"}
	StartTimeNextLatch AT %I* : ULINT;
END_STRUCT
END_TYPE

// ---- DUTs/IO/PDOs/AI_CycleCount_B1A935A2.TcDUT
{attribute 'GeneratedUsingTerminal: EL3773-0000-0016'}
{attribute addProperty BoxType "EL3773-0000-0016"}
{attribute addProperty Id "Cycle_CountAT %I*UINT2"}
{attribute addProperty CRC "2980656546"}
{attribute addProperty Size "2"}
TYPE AI_CycleCount_B1A935A2 EXTENDS InputBase_8311D824 :
STRUCT
	{attribute addProperty Name "Cycle_Count"}
	Cycle_Count AT %I* : UINT;
END_STRUCT
END_TYPE

// ---- DUTs/IO/PDOs/InfoData_BEF6B88E.TcDUT
{attribute 'GeneratedUsingTerminal: EL3773-0000-0016'}
{attribute addProperty BoxType "EL3773-0000-0016"}
{attribute addProperty Id "AdsAddrAT %I*AMSADDR8DcOutputShiftAT %I*DINT4DcInputShiftAT %I*DINT4StateAT %I*UINT2"}
{attribute addProperty CRC "3203840142"}
{attribute addProperty Size "18"}
TYPE InfoData_BEF6B88E EXTENDS InputBase_8311D824 :
STRUCT
	{attribute addProperty Name "AdsAddr"}
	AdsAddr AT %I* : AMSADDR;
	{attribute addProperty Name "DcOutputShift"}
	DcOutputShift AT %I* : DINT;
	{attribute addProperty Name "DcInputShift"}
	DcInputShift AT %I* : DINT;
	{attribute addProperty Name "State"}
	State AT %I* : UINT;
END_STRUCT
END_TYPE

// ---- DUTs/IO/PDOs/Digital_BD004D6F.TcDUT
{attribute 'GeneratedUsingTerminal: EM7004-0000-9995'}
{attribute addProperty BoxType "EM7004-0000-9995"}
{attribute addProperty Id "InputAT %I*ARRAY[0..15] OF BOOL16"}
{attribute addProperty CRC "2621435360"}
{attribute addProperty Size "16"}
TYPE Digital_BD004D6F EXTENDS InputBase_8311D824 :
STRUCT
	{attribute addProperty Name "Input"}
	Input AT %I* : ARRAY[0..15] OF BOOL;
END_STRUCT
END_TYPE

// ---- DUTs/IO/PDOs/Encoder_Channel_2E4EA213.TcDUT
{attribute 'GeneratedUsingTerminal: EM7004-0000-9995'}
{attribute addProperty BoxType "EM7004-0000-9995"}
{attribute addProperty Id "StatusAT %I*UINT2ValueAT %I*UINT2LatchAT %I*UINT2"}
{attribute addProperty CRC "776905235"}
{attribute addProperty Size "6"}
TYPE Encoder_Channel_2E4EA213 EXTENDS InputBase_8311D824 :
STRUCT
	{attribute addProperty Name "Status"}
	Status AT %I* : UINT;
	{attribute addProperty Name "Value"}
	Value AT %I* : UINT;
	{attribute addProperty Name "Latch"}
	Latch AT %I* : UINT;
END_STRUCT
END_TYPE

// ---- DUTs/IO/PDOs/Digital_A7E1DFAB.TcDUT
{attribute 'GeneratedUsingTerminal: EM7004-0000-9995'}
{attribute addProperty BoxType "EM7004-0000-9995"}
{attribute addProperty Id "OutputAT %Q*ARRAY[0..15] OF BOOL16"}
{attribute addProperty CRC "1538723034"}
{attribute addProperty Size "16"}
TYPE Digital_A7E1DFAB EXTENDS OutputBase_10CEE7DE :
STRUCT
	{attribute addProperty Name "Output"}
	Output AT %Q* : ARRAY[0..15] OF BOOL;
END_STRUCT
END_TYPE

// ---- DUTs/IO/PDOs/Analog_Channel_5F9B7EA6.TcDUT
{attribute 'GeneratedUsingTerminal: EM7004-0000-9995'}
{attribute addProperty BoxType "EM7004-0000-9995"}
{attribute addProperty Id "OutputAT %Q*INT2"}
{attribute addProperty CRC "1604026022"}
{attribute addProperty Size "2"}
TYPE Analog_Channel_5F9B7EA6 EXTENDS OutputBase_10CEE7DE :
STRUCT
	{attribute addProperty Name "Output"}
	Output AT %Q* : INT;
END_STRUCT
END_TYPE

// ---- DUTs/IO/PDOs/Encoder_Channel_B7999E14.TcDUT
{attribute 'GeneratedUsingTerminal: EM7004-0000-9995'}
{attribute addProperty BoxType "EM7004-0000-9995"}
{attribute addProperty Id "CtrlAT %Q*UINT2ValueAT %Q*UINT2"}
{attribute addProperty CRC "3080298004"}
{attribute addProperty Size "4"}
TYPE Encoder_Channel_B7999E14 EXTENDS OutputBase_10CEE7DE :
STRUCT
	{attribute addProperty Name "Ctrl"}
	Ctrl AT %Q* : UINT;
	{attribute addProperty Name "Value"}
	Value AT %Q* : UINT;
END_STRUCT
END_TYPE

// ---- DUTs/IO/PDOs/DeviceMain_Outputs_650F3486.TcDUT
{attribute 'GeneratedUsingTerminal: AX8108-0100-0101-0101'}
{attribute addProperty BoxType "AX8108-0100-0101-0101"}
{attribute addProperty Id "Power_supply_controlwordAT %Q*UINT2"}
{attribute addProperty CRC "1695495302"}
{attribute addProperty Size "2"}
TYPE DeviceMain_Outputs_650F3486 EXTENDS OutputBase_10CEE7DE :
STRUCT
	{attribute addProperty Name "Power_supply_controlword"}
	Power_supply_controlword AT %Q* : UINT;
END_STRUCT
END_TYPE

// ---- DUTs/IO/PDOs/FSoE_Slave_Connection_1_Slave_Message_330A35E4.TcDUT
{attribute 'GeneratedUsingTerminal: AX8108-0100-0101-0101'}
{attribute addProperty BoxType "AX8108-0100-0101-0101"}
{attribute addProperty Id "FSOEAT %I*FSOE_31BB7F2A21"}
{attribute addProperty CRC "856307172"}
{attribute addProperty Size "21"}
TYPE FSoE_Slave_Connection_1_Slave_Message_330A35E4 EXTENDS InputBase_8311D824 :
STRUCT
	{attribute addProperty Name "FSOE"}
	FSOE AT %I* : FSOE_31BB7F2A;
END_STRUCT
END_TYPE

// ---- DUTs/IO/PDOs/Standard_Inputdata_FDD1436A.TcDUT
{attribute 'GeneratedUsingTerminal: AX8108-0100-0101-0101'}
{attribute addProperty BoxType "AX8108-0100-0101-0101"}
{attribute addProperty Id "FSOEAT %I*FSOE_3C294B218"}
{attribute addProperty CRC "4258349930"}
{attribute addProperty Size "8"}
TYPE Standard_Inputdata_FDD1436A EXTENDS InputBase_8311D824 :
STRUCT
	{attribute addProperty Name "FSOE"}
	FSOE AT %I* : FSOE_3C294B21;
END_STRUCT
END_TYPE

// ---- DUTs/IO/PDOs/FSLOGIC_Inputs_CD3F9A93.TcDUT
{attribute 'GeneratedUsingTerminal: AX8108-0100-0101-0101'}
{attribute addProperty BoxType "AX8108-0100-0101-0101"}
{attribute addProperty Id "FSOEAT %I*FSOE_13BCEA3F2"}
{attribute addProperty CRC "3443497619"}
{attribute addProperty Size "2"}
TYPE FSLOGIC_Inputs_CD3F9A93 EXTENDS InputBase_8311D824 :
STRUCT
	{attribute addProperty Name "FSOE"}
	FSOE AT %I* : FSOE_13BCEA3F;
END_STRUCT
END_TYPE

// ---- DUTs/IO/PDOs/FSoE_Slave_Connection_1_Master_Message_7109E4F0.TcDUT
{attribute 'GeneratedUsingTerminal: AX8108-0100-0101-0101'}
{attribute addProperty BoxType "AX8108-0100-0101-0101"}
{attribute addProperty Id "FSOEAT %Q*FSOE_6A82EB9321"}
{attribute addProperty CRC "1896473840"}
{attribute addProperty Size "21"}
TYPE FSoE_Slave_Connection_1_Master_Message_7109E4F0 EXTENDS OutputBase_10CEE7DE :
STRUCT
	{attribute addProperty Name "FSOE"}
	FSOE AT %Q* : FSOE_6A82EB93;
END_STRUCT
END_TYPE

// ---- DUTs/IO/PDOs/Standard_Outputdata_59C030BE.TcDUT
{attribute 'GeneratedUsingTerminal: AX8108-0100-0101-0101'}
{attribute addProperty BoxType "AX8108-0100-0101-0101"}
{attribute addProperty Id "FSOEAT %Q*FSOE_BB3344D68"}
{attribute addProperty CRC "1505767614"}
{attribute addProperty Size "8"}
TYPE Standard_Outputdata_59C030BE EXTENDS OutputBase_10CEE7DE :
STRUCT
	{attribute addProperty Name "FSOE"}
	FSOE AT %Q* : FSOE_BB3344D6;
END_STRUCT
END_TYPE

// ---- DUTs/IO/PDOs/Ch_A_AxisMain_Inputs_DC14661D.TcDUT
{attribute 'GeneratedUsingTerminal: AX8108-0100-0101-0101'}
{attribute addProperty BoxType "AX8108-0100-0101-0101"}
{attribute addProperty Id "Ch_A_Position_actual_value_invalidAT %I*BOOL1Ch_A_1st_Additional_position_actual_value_invalidAT %I*BOOL1Ch_A_StatuswordAT %I*UINT2Ch_A_Position_actual_valueAT %I*DINT4"}
{attribute addProperty CRC "3692324381"}
{attribute addProperty Size "8"}
TYPE Ch_A_AxisMain_Inputs_DC14661D EXTENDS InputBase_8311D824 :
STRUCT
	{attribute addProperty Name "Ch_A_Position_actual_value_invalid"}
	Ch_A_Position_actual_value_invalid AT %I* : BOOL;
	{attribute addProperty Name "Ch_A_1st_Additional_position_actual_value_invalid"}
	Ch_A_1st_Additional_position_actual_value_invalid AT %I* : BOOL;
	{attribute addProperty Name "Ch_A_Statusword"}
	Ch_A_Statusword AT %I* : UINT;
	{attribute addProperty Name "Ch_A_Position_actual_value"}
	Ch_A_Position_actual_value AT %I* : DINT;
END_STRUCT
END_TYPE

// ---- DUTs/IO/PDOs/Ch_A_AxisMain_Outputs_A99AE12E.TcDUT
{attribute 'GeneratedUsingTerminal: AX8108-0100-0101-0101'}
{attribute addProperty BoxType "AX8108-0100-0101-0101"}
{attribute addProperty Id "Ch_A_ControlwordAT %Q*UINT2"}
{attribute addProperty CRC "2845499694"}
{attribute addProperty Size "2"}
TYPE Ch_A_AxisMain_Outputs_A99AE12E EXTENDS OutputBase_10CEE7DE :
STRUCT
	{attribute addProperty Name "Ch_A_Controlword"}
	Ch_A_Controlword AT %Q* : UINT;
END_STRUCT
END_TYPE

// ---- DUTs/IO/PDOs/Ch_A_Interpolator_Outputs_462A5F1D.TcDUT
{attribute 'GeneratedUsingTerminal: AX8108-0100-0101-0101'}
{attribute addProperty BoxType "AX8108-0100-0101-0101"}
{attribute addProperty Id "Ch_A_Target_positionAT %Q*DINT4Ch_A_Target_velocityAT %Q*DINT4"}
{attribute addProperty CRC "1177181981"}
{attribute addProperty Size "8"}
TYPE Ch_A_Interpolator_Outputs_462A5F1D EXTENDS OutputBase_10CEE7DE :
STRUCT
	{attribute addProperty Name "Ch_A_Target_position"}
	Ch_A_Target_position AT %Q* : DINT;
	{attribute addProperty Name "Ch_A_Target_velocity"}
	Ch_A_Target_velocity AT %Q* : DINT;
END_STRUCT
END_TYPE

// ---- DUTs/IO/PDOs/Ch_A_PositionControl_Inputs_8CB0F55A.TcDUT
{attribute 'GeneratedUsingTerminal: AX8108-0100-0101-0101'}
{attribute addProperty BoxType "AX8108-0100-0101-0101"}
{attribute addProperty Id "Ch_A_Following_error_actual_valueAT %I*DINT4"}
{attribute addProperty CRC "2360407386"}
{attribute addProperty Size "4"}
TYPE Ch_A_PositionControl_Inputs_8CB0F55A EXTENDS InputBase_8311D824 :
STRUCT
	{attribute addProperty Name "Ch_A_Following_error_actual_value"}
	Ch_A_Following_error_actual_value AT %I* : DINT;
END_STRUCT
END_TYPE

// ---- DUTs/IO/PDOs/WcState_B516A264.TcDUT
{attribute 'GeneratedUsingTerminal: AX8108-0100-0101-0101'}
{attribute addProperty BoxType "AX8108-0100-0101-0101"}
{attribute addProperty Id "WcState0AT %I*BOOL1WcState1AT %I*BOOL1InputToggle0AT %I*BOOL1InputToggle1AT %I*BOOL1"}
{attribute addProperty CRC "3038159460"}
{attribute addProperty Size "4"}
TYPE WcState_B516A264 EXTENDS InputBase_8311D824 :
STRUCT
	{attribute addProperty Name "WcState0"}
	WcState0 AT %I* : BOOL;
	{attribute addProperty Name "WcState1"}
	WcState1 AT %I* : BOOL;
	{attribute addProperty Name "InputToggle0"}
	InputToggle0 AT %I* : BOOL;
	{attribute addProperty Name "InputToggle1"}
	InputToggle1 AT %I* : BOOL;
END_STRUCT
END_TYPE

// ---- DUTs/IO/PDOs/InfoData_358A59CF.TcDUT
{attribute 'GeneratedUsingTerminal: AX8108-0100-0101-0101'}
{attribute addProperty BoxType "AX8108-0100-0101-0101"}
{attribute addProperty Id "AdsAddrAT %I*AMSADDR8DcOutputShiftAT %I*DINT4DcInputShiftAT %I*DINT4AoeNetIdAT %I*AMSNETID6Chn0AT %I*USINT1StateAT %I*UINT2"}
{attribute addProperty CRC "898259407"}
{attribute addProperty Size "25"}
TYPE InfoData_358A59CF EXTENDS InputBase_8311D824 :
STRUCT
	{attribute addProperty Name "AdsAddr"}
	AdsAddr AT %I* : AMSADDR;
	{attribute addProperty Name "DcOutputShift"}
	DcOutputShift AT %I* : DINT;
	{attribute addProperty Name "DcInputShift"}
	DcInputShift AT %I* : DINT;
	{attribute addProperty Name "AoeNetId"}
	AoeNetId AT %I* : AMSNETID;
	{attribute addProperty Name "Chn0"}
	Chn0 AT %I* : USINT;
	{attribute addProperty Name "State"}
	State AT %I* : UINT;
END_STRUCT
END_TYPE

// ---- DUTs/IO/PDOs/Device_6E257577.TcDUT
{attribute 'GeneratedUsingTerminal: AX8108-0100-0101-0101'}
{attribute addProperty BoxType "AX8108-0100-0101-0101"}
{attribute addProperty Id "DeviceMain_OutputsDeviceMain_Outputs_650F34862"}
{attribute addProperty CRC "1847948663"}
{attribute addProperty Size "2"}
TYPE Device_6E257577 :
STRUCT
	{attribute addProperty Name "DeviceMain_Outputs"}
	DeviceMain_Outputs  : DeviceMain_Outputs_650F3486;
END_STRUCT
END_TYPE

// ---- DUTs/IO/PDOs/Device_Safety_C21945A1.TcDUT
{attribute 'GeneratedUsingTerminal: AX8108-0100-0101-0101'}
{attribute addProperty BoxType "AX8108-0100-0101-0101"}
{attribute addProperty Id "FSoE_Slave_Connection_1_Slave_MessageFSoE_Slave_Connection_1_Slave_Message_330A35E421Standard_InputdataStandard_Inputdata_FDD1436A8FSLOGIC_InputsFSLOGIC_Inputs_CD3F9A932FSoE_Slave_Connection_1_Master_MessageFSoE_Slave_Connection_1_Master_Message_7109E4F021Standard_OutputdataStandard_Outputdata_59C030BE8FSLOGIC_OutputsEMPTY_STRUCTURE0"}
{attribute addProperty CRC "3256436129"}
{attribute addProperty Size "60"}
TYPE Device_Safety_C21945A1 :
STRUCT
	{attribute addProperty Name "FSoE_Slave_Connection_1_Slave_Message"}
	FSoE_Slave_Connection_1_Slave_Message  : FSoE_Slave_Connection_1_Slave_Message_330A35E4;
	{attribute addProperty Name "Standard_Inputdata"}
	Standard_Inputdata  : Standard_Inputdata_FDD1436A;
	{attribute addProperty Name "FSLOGIC_Inputs"}
	FSLOGIC_Inputs  : FSLOGIC_Inputs_CD3F9A93;
	{attribute addProperty Name "FSoE_Slave_Connection_1_Master_Message"}
	FSoE_Slave_Connection_1_Master_Message  : FSoE_Slave_Connection_1_Master_Message_7109E4F0;
	{attribute addProperty Name "Standard_Outputdata"}
	Standard_Outputdata  : Standard_Outputdata_59C030BE;
	{attribute addProperty Name "FSLOGIC_Outputs"}
	FSLOGIC_Outputs  : EMPTY_STRUCTURE;
END_STRUCT
END_TYPE

// ---- DUTs/IO/PDOs/Ch_A_1FF86D85.TcDUT
{attribute 'GeneratedUsingTerminal: AX8108-0100-0101-0101'}
{attribute addProperty BoxType "AX8108-0100-0101-0101"}
{attribute addProperty Id "Ch_A_AxisMain_InputsCh_A_AxisMain_Inputs_DC14661D8Ch_A_AxisMain_OutputsCh_A_AxisMain_Outputs_A99AE12E2Ch_A_Interpolator_OutputsCh_A_Interpolator_Outputs_462A5F1D8Ch_A_PositionControl_InputsCh_A_PositionControl_Inputs_8CB0F55A4"}
{attribute addProperty CRC "536374661"}
{attribute addProperty Size "22"}
TYPE Ch_A_1FF86D85 :
STRUCT
	{attribute addProperty Name "Ch_A_AxisMain_Inputs"}
	Ch_A_AxisMain_Inputs  : Ch_A_AxisMain_Inputs_DC14661D;
	{attribute addProperty Name "Ch_A_AxisMain_Outputs"}
	Ch_A_AxisMain_Outputs  : Ch_A_AxisMain_Outputs_A99AE12E;
	{attribute addProperty Name "Ch_A_Interpolator_Outputs"}
	Ch_A_Interpolator_Outputs  : Ch_A_Interpolator_Outputs_462A5F1D;
	{attribute addProperty Name "Ch_A_PositionControl_Inputs"}
	Ch_A_PositionControl_Inputs  : Ch_A_PositionControl_Inputs_8CB0F55A;
END_STRUCT
END_TYPE

// ---- DUTs/IO/PDOs/Ch_A_AxisMain_Inputs_BA7CE8DB.TcDUT
{attribute 'GeneratedUsingTerminal: AX8108-0100-0102-0102'}
{attribute addProperty BoxType "AX8108-0100-0102-0102"}
{attribute addProperty Id "Position_actual_value_invalidAT %I*BOOL1_1st_Additional_position_actual_value_invalidAT %I*BOOL1Ch_A_StatuswordAT %I*UINT2Ch_A_Position_actual_valueAT %I*DINT4"}
{attribute addProperty CRC "3128748251"}
{attribute addProperty Size "8"}
TYPE Ch_A_AxisMain_Inputs_BA7CE8DB EXTENDS InputBase_8311D824 :
STRUCT
	{attribute addProperty Name "Position_actual_value_invalid"}
	Position_actual_value_invalid AT %I* : BOOL;
	{attribute addProperty Name "_1st_Additional_position_actual_value_invalid"}
	_1st_Additional_position_actual_value_invalid AT %I* : BOOL;
	{attribute addProperty Name "Ch_A_Statusword"}
	Ch_A_Statusword AT %I* : UINT;
	{attribute addProperty Name "Ch_A_Position_actual_value"}
	Ch_A_Position_actual_value AT %I* : DINT;
END_STRUCT
END_TYPE

// ---- DUTs/IO/PDOs/Ch_A_D18C6F16.TcDUT
{attribute 'GeneratedUsingTerminal: AX8108-0100-0102-0102'}
{attribute addProperty BoxType "AX8108-0100-0102-0102"}
{attribute addProperty Id "Ch_A_AxisMain_InputsCh_A_AxisMain_Inputs_BA7CE8DB8Ch_A_AxisMain_OutputsCh_A_AxisMain_Outputs_A99AE12E2Ch_A_Interpolator_OutputsCh_A_Interpolator_Outputs_462A5F1D8Ch_A_PositionControl_InputsCh_A_PositionControl_Inputs_8CB0F55A4"}
{attribute addProperty CRC "3515641622"}
{attribute addProperty Size "22"}
TYPE Ch_A_D18C6F16 :
STRUCT
	{attribute addProperty Name "Ch_A_AxisMain_Inputs"}
	Ch_A_AxisMain_Inputs  : Ch_A_AxisMain_Inputs_BA7CE8DB;
	{attribute addProperty Name "Ch_A_AxisMain_Outputs"}
	Ch_A_AxisMain_Outputs  : Ch_A_AxisMain_Outputs_A99AE12E;
	{attribute addProperty Name "Ch_A_Interpolator_Outputs"}
	Ch_A_Interpolator_Outputs  : Ch_A_Interpolator_Outputs_462A5F1D;
	{attribute addProperty Name "Ch_A_PositionControl_Inputs"}
	Ch_A_PositionControl_Inputs  : Ch_A_PositionControl_Inputs_8CB0F55A;
END_STRUCT
END_TYPE

// ---- DUTs/IO/PDOs/Ch_B_AxisMain_Inputs_A10B23CB.TcDUT
{attribute 'GeneratedUsingTerminal: AX8206-0100-0101-0101'}
{attribute addProperty BoxType "AX8206-0100-0101-0101"}
{attribute addProperty Id "Ch_B_Position_actual_value_invalidAT %I*BOOL1Ch_B_1st_Additional_position_actual_value_invalidAT %I*BOOL1Ch_B_StatuswordAT %I*UINT2Ch_B_Position_actual_valueAT %I*DINT4"}
{attribute addProperty CRC "2701861835"}
{attribute addProperty Size "8"}
TYPE Ch_B_AxisMain_Inputs_A10B23CB EXTENDS InputBase_8311D824 :
STRUCT
	{attribute addProperty Name "Ch_B_Position_actual_value_invalid"}
	Ch_B_Position_actual_value_invalid AT %I* : BOOL;
	{attribute addProperty Name "Ch_B_1st_Additional_position_actual_value_invalid"}
	Ch_B_1st_Additional_position_actual_value_invalid AT %I* : BOOL;
	{attribute addProperty Name "Ch_B_Statusword"}
	Ch_B_Statusword AT %I* : UINT;
	{attribute addProperty Name "Ch_B_Position_actual_value"}
	Ch_B_Position_actual_value AT %I* : DINT;
END_STRUCT
END_TYPE

// ---- DUTs/IO/PDOs/Ch_B_AxisMain_Outputs_526A47F8.TcDUT
{attribute 'GeneratedUsingTerminal: AX8206-0100-0101-0101'}
{attribute addProperty BoxType "AX8206-0100-0101-0101"}
{attribute addProperty Id "Ch_B_ControlwordAT %Q*UINT2"}
{attribute addProperty CRC "1382696952"}
{attribute addProperty Size "2"}
TYPE Ch_B_AxisMain_Outputs_526A47F8 EXTENDS OutputBase_10CEE7DE :
STRUCT
	{attribute addProperty Name "Ch_B_Controlword"}
	Ch_B_Controlword AT %Q* : UINT;
END_STRUCT
END_TYPE

// ---- DUTs/IO/PDOs/Ch_B_Interpolator_Outputs_F819AE72.TcDUT
{attribute 'GeneratedUsingTerminal: AX8206-0100-0101-0101'}
{attribute addProperty BoxType "AX8206-0100-0101-0101"}
{attribute addProperty Id "Ch_B_Target_positionAT %Q*DINT4Ch_B_Target_velocityAT %Q*DINT4"}
{attribute addProperty CRC "4162432626"}
{attribute addProperty Size "8"}
TYPE Ch_B_Interpolator_Outputs_F819AE72 EXTENDS OutputBase_10CEE7DE :
STRUCT
	{attribute addProperty Name "Ch_B_Target_position"}
	Ch_B_Target_position AT %Q* : DINT;
	{attribute addProperty Name "Ch_B_Target_velocity"}
	Ch_B_Target_velocity AT %Q* : DINT;
END_STRUCT
END_TYPE

// ---- DUTs/IO/PDOs/Ch_B_PositionControl_Inputs_C884000A.TcDUT
{attribute 'GeneratedUsingTerminal: AX8206-0100-0101-0101'}
{attribute addProperty BoxType "AX8206-0100-0101-0101"}
{attribute addProperty Id "Ch_B_Following_error_actual_valueAT %I*DINT4"}
{attribute addProperty CRC "3364093962"}
{attribute addProperty Size "4"}
TYPE Ch_B_PositionControl_Inputs_C884000A EXTENDS InputBase_8311D824 :
STRUCT
	{attribute addProperty Name "Ch_B_Following_error_actual_value"}
	Ch_B_Following_error_actual_value AT %I* : DINT;
END_STRUCT
END_TYPE

// ---- DUTs/IO/PDOs/InfoData_386C00A5.TcDUT
{attribute 'GeneratedUsingTerminal: AX8206-0100-0101-0101'}
{attribute addProperty BoxType "AX8206-0100-0101-0101"}
{attribute addProperty Id "AdsAddrAT %I*AMSADDR8DcOutputShiftAT %I*DINT4DcInputShiftAT %I*DINT4AoeNetIdAT %I*AMSNETID6Chn0AT %I*USINT1Chn1AT %I*USINT1StateAT %I*UINT2"}
{attribute addProperty CRC "946602149"}
{attribute addProperty Size "26"}
TYPE InfoData_386C00A5 EXTENDS InputBase_8311D824 :
STRUCT
	{attribute addProperty Name "AdsAddr"}
	AdsAddr AT %I* : AMSADDR;
	{attribute addProperty Name "DcOutputShift"}
	DcOutputShift AT %I* : DINT;
	{attribute addProperty Name "DcInputShift"}
	DcInputShift AT %I* : DINT;
	{attribute addProperty Name "AoeNetId"}
	AoeNetId AT %I* : AMSNETID;
	{attribute addProperty Name "Chn0"}
	Chn0 AT %I* : USINT;
	{attribute addProperty Name "Chn1"}
	Chn1 AT %I* : USINT;
	{attribute addProperty Name "State"}
	State AT %I* : UINT;
END_STRUCT
END_TYPE

// ---- DUTs/IO/PDOs/Ch_B_5E084BAA.TcDUT
{attribute 'GeneratedUsingTerminal: AX8206-0100-0101-0101'}
{attribute addProperty BoxType "AX8206-0100-0101-0101"}
{attribute addProperty Id "Ch_B_AxisMain_InputsCh_B_AxisMain_Inputs_A10B23CB8Ch_B_AxisMain_OutputsCh_B_AxisMain_Outputs_526A47F82Ch_B_Interpolator_OutputsCh_B_Interpolator_Outputs_F819AE728Ch_B_PositionControl_InputsCh_B_PositionControl_Inputs_C884000A4"}
{attribute addProperty CRC "1577601962"}
{attribute addProperty Size "22"}
TYPE Ch_B_5E084BAA :
STRUCT
	{attribute addProperty Name "Ch_B_AxisMain_Inputs"}
	Ch_B_AxisMain_Inputs  : Ch_B_AxisMain_Inputs_A10B23CB;
	{attribute addProperty Name "Ch_B_AxisMain_Outputs"}
	Ch_B_AxisMain_Outputs  : Ch_B_AxisMain_Outputs_526A47F8;
	{attribute addProperty Name "Ch_B_Interpolator_Outputs"}
	Ch_B_Interpolator_Outputs  : Ch_B_Interpolator_Outputs_F819AE72;
	{attribute addProperty Name "Ch_B_PositionControl_Inputs"}
	Ch_B_PositionControl_Inputs  : Ch_B_PositionControl_Inputs_C884000A;
END_STRUCT
END_TYPE

// ---- DUTs/IO/PDOs/Ch_B_AxisMain_Inputs_3D4AF970.TcDUT
{attribute 'GeneratedUsingTerminal: AX8206-0100-0102-0102'}
{attribute addProperty BoxType "AX8206-0100-0102-0102"}
{attribute addProperty Id "Position_actual_value_invalidAT %I*BOOL1_1st_Additional_position_actual_value_invalidAT %I*BOOL1Ch_B_StatuswordAT %I*UINT2Ch_B_Position_actual_valueAT %I*DINT4"}
{attribute addProperty CRC "1028323696"}
{attribute addProperty Size "8"}
TYPE Ch_B_AxisMain_Inputs_3D4AF970 EXTENDS InputBase_8311D824 :
STRUCT
	{attribute addProperty Name "Position_actual_value_invalid"}
	Position_actual_value_invalid AT %I* : BOOL;
	{attribute addProperty Name "_1st_Additional_position_actual_value_invalid"}
	_1st_Additional_position_actual_value_invalid AT %I* : BOOL;
	{attribute addProperty Name "Ch_B_Statusword"}
	Ch_B_Statusword AT %I* : UINT;
	{attribute addProperty Name "Ch_B_Position_actual_value"}
	Ch_B_Position_actual_value AT %I* : DINT;
END_STRUCT
END_TYPE

// ---- DUTs/IO/PDOs/Ch_B_647F9A0C.TcDUT
{attribute 'GeneratedUsingTerminal: AX8206-0100-0102-0102'}
{attribute addProperty BoxType "AX8206-0100-0102-0102"}
{attribute addProperty Id "Ch_B_AxisMain_InputsCh_B_AxisMain_Inputs_3D4AF9708Ch_B_AxisMain_OutputsCh_B_AxisMain_Outputs_526A47F82Ch_B_Interpolator_OutputsCh_B_Interpolator_Outputs_F819AE728Ch_B_PositionControl_InputsCh_B_PositionControl_Inputs_C884000A4"}
{attribute addProperty CRC "1686084108"}
{attribute addProperty Size "22"}
TYPE Ch_B_647F9A0C :
STRUCT
	{attribute addProperty Name "Ch_B_AxisMain_Inputs"}
	Ch_B_AxisMain_Inputs  : Ch_B_AxisMain_Inputs_3D4AF970;
	{attribute addProperty Name "Ch_B_AxisMain_Outputs"}
	Ch_B_AxisMain_Outputs  : Ch_B_AxisMain_Outputs_526A47F8;
	{attribute addProperty Name "Ch_B_Interpolator_Outputs"}
	Ch_B_Interpolator_Outputs  : Ch_B_Interpolator_Outputs_F819AE72;
	{attribute addProperty Name "Ch_B_PositionControl_Inputs"}
	Ch_B_PositionControl_Inputs  : Ch_B_PositionControl_Inputs_C884000A;
END_STRUCT
END_TYPE

// ---- DUTs/IO/PDOs/InfoData_E68C61CD.TcDUT
{attribute 'GeneratedUsingTerminal: IODEVICETYPE_ETHERCATPROT'}
{attribute addProperty BoxType "IODEVICETYPE_ETHERCATPROT"}
{attribute addProperty Id "ChangeCountAT %I*UINT2DevIdAT %I*UINT2AmsNetIdAT %I*AMSNETID6CfgSlaveCountAT %I*UINT2DcToTcTimeOffsetAT %I*LINT8DcToExtTimeOffsetAT %I*LINT8"}
{attribute addProperty CRC "3867959757"}
{attribute addProperty Size "28"}
TYPE InfoData_E68C61CD EXTENDS InputBase_8311D824 :
STRUCT
	{attribute addProperty Name "ChangeCount"}
	ChangeCount AT %I* : UINT;
	{attribute addProperty Name "DevId"}
	DevId AT %I* : UINT;
	{attribute addProperty Name "AmsNetId"}
	AmsNetId AT %I* : AMSNETID;
	{attribute addProperty Name "CfgSlaveCount"}
	CfgSlaveCount AT %I* : UINT;
	{attribute addProperty Name "DcToTcTimeOffset"}
	DcToTcTimeOffset AT %I* : LINT;
	{attribute addProperty Name "DcToExtTimeOffset"}
	DcToExtTimeOffset AT %I* : LINT;
END_STRUCT
END_TYPE

// ---- DUTs/IO/PDOs/InfoData_2A97D6CF.TcDUT
{attribute 'GeneratedUsingTerminal: IODEVICETYPE_ETHERCATPROT'}
{attribute addProperty BoxType "IODEVICETYPE_ETHERCATPROT"}
{attribute addProperty Id "ObjectIdAT %I*OTCID4StateAT %I*UINT2SlaveCountAT %I*UINT2"}
{attribute addProperty CRC "714593999"}
{attribute addProperty Size "8"}
TYPE InfoData_2A97D6CF EXTENDS InputBase_8311D824 :
STRUCT
	{attribute addProperty Name "ObjectId"}
	ObjectId AT %I* : OTCID;
	{attribute addProperty Name "State"}
	State AT %I* : UINT;
	{attribute addProperty Name "SlaveCount"}
	SlaveCount AT %I* : UINT;
END_STRUCT
END_TYPE

// ---- DUTs/IO/PDOs/Inputs_25A0042B.TcDUT
{attribute 'GeneratedUsingTerminal: IODEVICETYPE_ETHERCATPROT'}
{attribute addProperty BoxType "IODEVICETYPE_ETHERCATPROT"}
{attribute addProperty Id "SlaveCountAT %I*UINT2DevStateAT %I*UINT2Frm0StateAT %I*UINT2Frm0WcStateAT %I*UINT2Frm0InputToggleAT %I*UINT2Frm1StateAT %I*UINT2Frm1WcStateAT %I*UINT2Frm1InputToggleAT %I*UINT2Frm2StateAT %I*UINT2Frm2WcStateAT %I*UINT2Frm2InputToggleAT %I*UINT2Frm3StateAT %I*UINT2Frm3WcStateAT %I*UINT2Frm3InputToggleAT %I*UINT2Frm4StateAT %I*UINT2Frm4WcStateAT %I*UINT2Frm4InputToggleAT %I*UINT2Frm5StateAT %I*UINT2Frm5WcStateAT %I*UINT2Frm5InputToggleAT %I*UINT2Frm6StateAT %I*UINT2Frm6WcStateAT %I*UINT2Frm6InputToggleAT %I*UINT2Frm7StateAT %I*UINT2Frm7WcStateAT %I*UINT2Frm7InputToggleAT %I*UINT2Frm8StateAT %I*UINT2Frm8WcStateAT %I*UINT2Frm8InputToggleAT %I*UINT2Frm9StateAT %I*UINT2Frm9WcStateAT %I*UINT2Frm9InputToggleAT %I*UINT2Frm10StateAT %I*UINT2Frm10WcStateAT %I*UINT2Frm10InputToggleAT %I*UINT2Frm11StateAT %I*UINT2Frm11WcStateAT %I*UINT2Frm11InputToggleAT %I*UINT2Frm12StateAT %I*UINT2Frm12WcStateAT %I*UINT2Frm12InputToggleAT %I*UINT2Frm13StateAT %I*UINT2Frm13WcStateAT %I*UINT2Frm13InputToggleAT %I*UINT2Frm14StateAT %I*UINT2Frm14WcStateAT %I*UINT2Frm14InputToggleAT %I*UINT2Frm15StateAT %I*UINT2Frm15WcStateAT %I*UINT2Frm15InputToggleAT %I*UINT2Frm16StateAT %I*UINT2Frm16WcStateAT %I*UINT2Frm16InputToggleAT %I*UINT2Frm17StateAT %I*UINT2Frm17WcStateAT %I*UINT2Frm17InputToggleAT %I*UINT2Frm18StateAT %I*UINT2Frm18WcStateAT %I*UINT2Frm18InputToggleAT %I*UINT2Frm19StateAT %I*UINT2Frm19WcStateAT %I*UINT2Frm19InputToggleAT %I*UINT2Frm20StateAT %I*UINT2Frm20WcStateAT %I*UINT2Frm20InputToggleAT %I*UINT2Frm21StateAT %I*UINT2Frm21WcStateAT %I*UINT2Frm21InputToggleAT %I*UINT2Frm22StateAT %I*UINT2Frm22WcStateAT %I*UINT2Frm22InputToggleAT %I*UINT2Frm23StateAT %I*UINT2Frm23WcStateAT %I*UINT2Frm23InputToggleAT %I*UINT2Frm24StateAT %I*UINT2Frm24WcStateAT %I*UINT2Frm24InputToggleAT %I*UINT2Frm25StateAT %I*UINT2Frm25WcStateAT %I*UINT2Frm25InputToggleAT %I*UINT2"}
{attribute addProperty CRC "631243819"}
{attribute addProperty Size "160"}
TYPE Inputs_25A0042B EXTENDS InputBase_8311D824 :
STRUCT
	{attribute addProperty Name "SlaveCount"}
	SlaveCount AT %I* : UINT;
	{attribute addProperty Name "DevState"}
	DevState AT %I* : UINT;
	{attribute addProperty Name "Frm0State"}
	Frm0State AT %I* : UINT;
	{attribute addProperty Name "Frm0WcState"}
	Frm0WcState AT %I* : UINT;
	{attribute addProperty Name "Frm0InputToggle"}
	Frm0InputToggle AT %I* : UINT;
	{attribute addProperty Name "Frm1State"}
	Frm1State AT %I* : UINT;
	{attribute addProperty Name "Frm1WcState"}
	Frm1WcState AT %I* : UINT;
	{attribute addProperty Name "Frm1InputToggle"}
	Frm1InputToggle AT %I* : UINT;
	{attribute addProperty Name "Frm2State"}
	Frm2State AT %I* : UINT;
	{attribute addProperty Name "Frm2WcState"}
	Frm2WcState AT %I* : UINT;
	{attribute addProperty Name "Frm2InputToggle"}
	Frm2InputToggle AT %I* : UINT;
	{attribute addProperty Name "Frm3State"}
	Frm3State AT %I* : UINT;
	{attribute addProperty Name "Frm3WcState"}
	Frm3WcState AT %I* : UINT;
	{attribute addProperty Name "Frm3InputToggle"}
	Frm3InputToggle AT %I* : UINT;
	{attribute addProperty Name "Frm4State"}
	Frm4State AT %I* : UINT;
	{attribute addProperty Name "Frm4WcState"}
	Frm4WcState AT %I* : UINT;
	{attribute addProperty Name "Frm4InputToggle"}
	Frm4InputToggle AT %I* : UINT;
	{attribute addProperty Name "Frm5State"}
	Frm5State AT %I* : UINT;
	{attribute addProperty Name "Frm5WcState"}
	Frm5WcState AT %I* : UINT;
	{attribute addProperty Name "Frm5InputToggle"}
	Frm5InputToggle AT %I* : UINT;
	{attribute addProperty Name "Frm6State"}
	Frm6State AT %I* : UINT;
	{attribute addProperty Name "Frm6WcState"}
	Frm6WcState AT %I* : UINT;
	{attribute addProperty Name "Frm6InputToggle"}
	Frm6InputToggle AT %I* : UINT;
	{attribute addProperty Name "Frm7State"}
	Frm7State AT %I* : UINT;
	{attribute addProperty Name "Frm7WcState"}
	Frm7WcState AT %I* : UINT;
	{attribute addProperty Name "Frm7InputToggle"}
	Frm7InputToggle AT %I* : UINT;
	{attribute addProperty Name "Frm8State"}
	Frm8State AT %I* : UINT;
	{attribute addProperty Name "Frm8WcState"}
	Frm8WcState AT %I* : UINT;
	{attribute addProperty Name "Frm8InputToggle"}
	Frm8InputToggle AT %I* : UINT;
	{attribute addProperty Name "Frm9State"}
	Frm9State AT %I* : UINT;
	{attribute addProperty Name "Frm9WcState"}
	Frm9WcState AT %I* : UINT;
	{attribute addProperty Name "Frm9InputToggle"}
	Frm9InputToggle AT %I* : UINT;
	{attribute addProperty Name "Frm10State"}
	Frm10State AT %I* : UINT;
	{attribute addProperty Name "Frm10WcState"}
	Frm10WcState AT %I* : UINT;
	{attribute addProperty Name "Frm10InputToggle"}
	Frm10InputToggle AT %I* : UINT;
	{attribute addProperty Name "Frm11State"}
	Frm11State AT %I* : UINT;
	{attribute addProperty Name "Frm11WcState"}
	Frm11WcState AT %I* : UINT;
	{attribute addProperty Name "Frm11InputToggle"}
	Frm11InputToggle AT %I* : UINT;
	{attribute addProperty Name "Frm12State"}
	Frm12State AT %I* : UINT;
	{attribute addProperty Name "Frm12WcState"}
	Frm12WcState AT %I* : UINT;
	{attribute addProperty Name "Frm12InputToggle"}
	Frm12InputToggle AT %I* : UINT;
	{attribute addProperty Name "Frm13State"}
	Frm13State AT %I* : UINT;
	{attribute addProperty Name "Frm13WcState"}
	Frm13WcState AT %I* : UINT;
	{attribute addProperty Name "Frm13InputToggle"}
	Frm13InputToggle AT %I* : UINT;
	{attribute addProperty Name "Frm14State"}
	Frm14State AT %I* : UINT;
	{attribute addProperty Name "Frm14WcState"}
	Frm14WcState AT %I* : UINT;
	{attribute addProperty Name "Frm14InputToggle"}
	Frm14InputToggle AT %I* : UINT;
	{attribute addProperty Name "Frm15State"}
	Frm15State AT %I* : UINT;
	{attribute addProperty Name "Frm15WcState"}
	Frm15WcState AT %I* : UINT;
	{attribute addProperty Name "Frm15InputToggle"}
	Frm15InputToggle AT %I* : UINT;
	{attribute addProperty Name "Frm16State"}
	Frm16State AT %I* : UINT;
	{attribute addProperty Name "Frm16WcState"}
	Frm16WcState AT %I* : UINT;
	{attribute addProperty Name "Frm16InputToggle"}
	Frm16InputToggle AT %I* : UINT;
	{attribute addProperty Name "Frm17State"}
	Frm17State AT %I* : UINT;
	{attribute addProperty Name "Frm17WcState"}
	Frm17WcState AT %I* : UINT;
	{attribute addProperty Name "Frm17InputToggle"}
	Frm17InputToggle AT %I* : UINT;
	{attribute addProperty Name "Frm18State"}
	Frm18State AT %I* : UINT;
	{attribute addProperty Name "Frm18WcState"}
	Frm18WcState AT %I* : UINT;
	{attribute addProperty Name "Frm18InputToggle"}
	Frm18InputToggle AT %I* : UINT;
	{attribute addProperty Name "Frm19State"}
	Frm19State AT %I* : UINT;
	{attribute addProperty Name "Frm19WcState"}
	Frm19WcState AT %I* : UINT;
	{attribute addProperty Name "Frm19InputToggle"}
	Frm19InputToggle AT %I* : UINT;
	{attribute addProperty Name "Frm20State"}
	Frm20State AT %I* : UINT;
	{attribute addProperty Name "Frm20WcState"}
	Frm20WcState AT %I* : UINT;
	{attribute addProperty Name "Frm20InputToggle"}
	Frm20InputToggle AT %I* : UINT;
	{attribute addProperty Name "Frm21State"}
	Frm21State AT %I* : UINT;
	{attribute addProperty Name "Frm21WcState"}
	Frm21WcState AT %I* : UINT;
	{attribute addProperty Name "Frm21InputToggle"}
	Frm21InputToggle AT %I* : UINT;
	{attribute addProperty Name "Frm22State"}
	Frm22State AT %I* : UINT;
	{attribute addProperty Name "Frm22WcState"}
	Frm22WcState AT %I* : UINT;
	{attribute addProperty Name "Frm22InputToggle"}
	Frm22InputToggle AT %I* : UINT;
	{attribute addProperty Name "Frm23State"}
	Frm23State AT %I* : UINT;
	{attribute addProperty Name "Frm23WcState"}
	Frm23WcState AT %I* : UINT;
	{attribute addProperty Name "Frm23InputToggle"}
	Frm23InputToggle AT %I* : UINT;
	{attribute addProperty Name "Frm24State"}
	Frm24State AT %I* : UINT;
	{attribute addProperty Name "Frm24WcState"}
	Frm24WcState AT %I* : UINT;
	{attribute addProperty Name "Frm24InputToggle"}
	Frm24InputToggle AT %I* : UINT;
	{attribute addProperty Name "Frm25State"}
	Frm25State AT %I* : UINT;
	{attribute addProperty Name "Frm25WcState"}
	Frm25WcState AT %I* : UINT;
	{attribute addProperty Name "Frm25InputToggle"}
	Frm25InputToggle AT %I* : UINT;
END_STRUCT
END_TYPE

// ---- DUTs/IO/PDOs/Outputs_2397A10E.TcDUT
{attribute 'GeneratedUsingTerminal: IODEVICETYPE_ETHERCATPROT'}
{attribute addProperty BoxType "IODEVICETYPE_ETHERCATPROT"}
{attribute addProperty Id "DevCtrlAT %Q*UINT2Frm0CtrlAT %Q*UINT2Frm0WcCtrlAT %Q*UINT2Frm1CtrlAT %Q*UINT2Frm1WcCtrlAT %Q*UINT2Frm2CtrlAT %Q*UINT2Frm2WcCtrlAT %Q*UINT2Frm3CtrlAT %Q*UINT2Frm3WcCtrlAT %Q*UINT2Frm4CtrlAT %Q*UINT2Frm4WcCtrlAT %Q*UINT2Frm5CtrlAT %Q*UINT2Frm5WcCtrlAT %Q*UINT2Frm6CtrlAT %Q*UINT2Frm6WcCtrlAT %Q*UINT2Frm7CtrlAT %Q*UINT2Frm7WcCtrlAT %Q*UINT2Frm8CtrlAT %Q*UINT2Frm8WcCtrlAT %Q*UINT2Frm9CtrlAT %Q*UINT2Frm9WcCtrlAT %Q*UINT2Frm10CtrlAT %Q*UINT2Frm10WcCtrlAT %Q*UINT2Frm11CtrlAT %Q*UINT2Frm11WcCtrlAT %Q*UINT2Frm12CtrlAT %Q*UINT2Frm12WcCtrlAT %Q*UINT2Frm13CtrlAT %Q*UINT2Frm13WcCtrlAT %Q*UINT2Frm14CtrlAT %Q*UINT2Frm14WcCtrlAT %Q*UINT2Frm15CtrlAT %Q*UINT2Frm15WcCtrlAT %Q*UINT2Frm16CtrlAT %Q*UINT2Frm16WcCtrlAT %Q*UINT2Frm17CtrlAT %Q*UINT2Frm17WcCtrlAT %Q*UINT2Frm18CtrlAT %Q*UINT2Frm18WcCtrlAT %Q*UINT2Frm19CtrlAT %Q*UINT2Frm19WcCtrlAT %Q*UINT2Frm20CtrlAT %Q*UINT2Frm20WcCtrlAT %Q*UINT2Frm21CtrlAT %Q*UINT2Frm21WcCtrlAT %Q*UINT2Frm22CtrlAT %Q*UINT2Frm22WcCtrlAT %Q*UINT2Frm23CtrlAT %Q*UINT2Frm23WcCtrlAT %Q*UINT2Frm24CtrlAT %Q*UINT2Frm24WcCtrlAT %Q*UINT2Frm25CtrlAT %Q*UINT2Frm25WcCtrlAT %Q*UINT2"}
{attribute addProperty CRC "597139726"}
{attribute addProperty Size "106"}
TYPE Outputs_2397A10E EXTENDS OutputBase_10CEE7DE :
STRUCT
	{attribute addProperty Name "DevCtrl"}
	DevCtrl AT %Q* : UINT;
	{attribute addProperty Name "Frm0Ctrl"}
	Frm0Ctrl AT %Q* : UINT;
	{attribute addProperty Name "Frm0WcCtrl"}
	Frm0WcCtrl AT %Q* : UINT;
	{attribute addProperty Name "Frm1Ctrl"}
	Frm1Ctrl AT %Q* : UINT;
	{attribute addProperty Name "Frm1WcCtrl"}
	Frm1WcCtrl AT %Q* : UINT;
	{attribute addProperty Name "Frm2Ctrl"}
	Frm2Ctrl AT %Q* : UINT;
	{attribute addProperty Name "Frm2WcCtrl"}
	Frm2WcCtrl AT %Q* : UINT;
	{attribute addProperty Name "Frm3Ctrl"}
	Frm3Ctrl AT %Q* : UINT;
	{attribute addProperty Name "Frm3WcCtrl"}
	Frm3WcCtrl AT %Q* : UINT;
	{attribute addProperty Name "Frm4Ctrl"}
	Frm4Ctrl AT %Q* : UINT;
	{attribute addProperty Name "Frm4WcCtrl"}
	Frm4WcCtrl AT %Q* : UINT;
	{attribute addProperty Name "Frm5Ctrl"}
	Frm5Ctrl AT %Q* : UINT;
	{attribute addProperty Name "Frm5WcCtrl"}
	Frm5WcCtrl AT %Q* : UINT;
	{attribute addProperty Name "Frm6Ctrl"}
	Frm6Ctrl AT %Q* : UINT;
	{attribute addProperty Name "Frm6WcCtrl"}
	Frm6WcCtrl AT %Q* : UINT;
	{attribute addProperty Name "Frm7Ctrl"}
	Frm7Ctrl AT %Q* : UINT;
	{attribute addProperty Name "Frm7WcCtrl"}
	Frm7WcCtrl AT %Q* : UINT;
	{attribute addProperty Name "Frm8Ctrl"}
	Frm8Ctrl AT %Q* : UINT;
	{attribute addProperty Name "Frm8WcCtrl"}
	Frm8WcCtrl AT %Q* : UINT;
	{attribute addProperty Name "Frm9Ctrl"}
	Frm9Ctrl AT %Q* : UINT;
	{attribute addProperty Name "Frm9WcCtrl"}
	Frm9WcCtrl AT %Q* : UINT;
	{attribute addProperty Name "Frm10Ctrl"}
	Frm10Ctrl AT %Q* : UINT;
	{attribute addProperty Name "Frm10WcCtrl"}
	Frm10WcCtrl AT %Q* : UINT;
	{attribute addProperty Name "Frm11Ctrl"}
	Frm11Ctrl AT %Q* : UINT;
	{attribute addProperty Name "Frm11WcCtrl"}
	Frm11WcCtrl AT %Q* : UINT;
	{attribute addProperty Name "Frm12Ctrl"}
	Frm12Ctrl AT %Q* : UINT;
	{attribute addProperty Name "Frm12WcCtrl"}
	Frm12WcCtrl AT %Q* : UINT;
	{attribute addProperty Name "Frm13Ctrl"}
	Frm13Ctrl AT %Q* : UINT;
	{attribute addProperty Name "Frm13WcCtrl"}
	Frm13WcCtrl AT %Q* : UINT;
	{attribute addProperty Name "Frm14Ctrl"}
	Frm14Ctrl AT %Q* : UINT;
	{attribute addProperty Name "Frm14WcCtrl"}
	Frm14WcCtrl AT %Q* : UINT;
	{attribute addProperty Name "Frm15Ctrl"}
	Frm15Ctrl AT %Q* : UINT;
	{attribute addProperty Name "Frm15WcCtrl"}
	Frm15WcCtrl AT %Q* : UINT;
	{attribute addProperty Name "Frm16Ctrl"}
	Frm16Ctrl AT %Q* : UINT;
	{attribute addProperty Name "Frm16WcCtrl"}
	Frm16WcCtrl AT %Q* : UINT;
	{attribute addProperty Name "Frm17Ctrl"}
	Frm17Ctrl AT %Q* : UINT;
	{attribute addProperty Name "Frm17WcCtrl"}
	Frm17WcCtrl AT %Q* : UINT;
	{attribute addProperty Name "Frm18Ctrl"}
	Frm18Ctrl AT %Q* : UINT;
	{attribute addProperty Name "Frm18WcCtrl"}
	Frm18WcCtrl AT %Q* : UINT;
	{attribute addProperty Name "Frm19Ctrl"}
	Frm19Ctrl AT %Q* : UINT;
	{attribute addProperty Name "Frm19WcCtrl"}
	Frm19WcCtrl AT %Q* : UINT;
	{attribute addProperty Name "Frm20Ctrl"}
	Frm20Ctrl AT %Q* : UINT;
	{attribute addProperty Name "Frm20WcCtrl"}
	Frm20WcCtrl AT %Q* : UINT;
	{attribute addProperty Name "Frm21Ctrl"}
	Frm21Ctrl AT %Q* : UINT;
	{attribute addProperty Name "Frm21WcCtrl"}
	Frm21WcCtrl AT %Q* : UINT;
	{attribute addProperty Name "Frm22Ctrl"}
	Frm22Ctrl AT %Q* : UINT;
	{attribute addProperty Name "Frm22WcCtrl"}
	Frm22WcCtrl AT %Q* : UINT;
	{attribute addProperty Name "Frm23Ctrl"}
	Frm23Ctrl AT %Q* : UINT;
	{attribute addProperty Name "Frm23WcCtrl"}
	Frm23WcCtrl AT %Q* : UINT;
	{attribute addProperty Name "Frm24Ctrl"}
	Frm24Ctrl AT %Q* : UINT;
	{attribute addProperty Name "Frm24WcCtrl"}
	Frm24WcCtrl AT %Q* : UINT;
	{attribute addProperty Name "Frm25Ctrl"}
	Frm25Ctrl AT %Q* : UINT;
	{attribute addProperty Name "Frm25WcCtrl"}
	Frm25WcCtrl AT %Q* : UINT;
END_STRUCT
END_TYPE

// ---- DUTs/IO/Boxes/EK1100_1FC0878B.TcDUT
{attribute 'GeneratedUsingTerminal: EK1100-0000-0018'}
{attribute addProperty BoxType "EK1100-0000-0018"}
{attribute addProperty Description "EK1100 EtherCAT Coupler (2A E-Bus)"}
{attribute addProperty Physics "YKY"}
{attribute addProperty Id "InfoDataAT %I*InfoData_6F19DB2B2"}
{attribute addProperty CRC "532711307"}
{attribute addProperty Size "2"}
TYPE EK1100_1FC0878B EXTENDS EtcSlaveBoxBase_77A0E4A7 :
STRUCT
	{attribute addProperty Name "InfoData"}
	InfoData : InfoData_6F19DB2B;
END_STRUCT
END_TYPE

// ---- DUTs/IO/Boxes/EK1122_1FC0878B.TcDUT
{attribute 'GeneratedUsingTerminal: EK1122-0000-0018'}
{attribute addProperty BoxType "EK1122-0000-0018"}
{attribute addProperty Description "EK1122 2 port EtherCAT junction"}
{attribute addProperty Physics "KYKY"}
{attribute addProperty Id "InfoDataAT %I*InfoData_6F19DB2B2"}
{attribute addProperty CRC "532711307"}
{attribute addProperty Size "2"}
TYPE EK1122_1FC0878B EXTENDS EtcSlaveTerminalBase_947E5A46 :
STRUCT
	{attribute addProperty Name "InfoData"}
	InfoData : InfoData_6F19DB2B;
END_STRUCT
END_TYPE

